# B&R Automation Studio project mappFramework (part 2)

### SimpleCfg.mpreportcore - PC/mappServices/Report/SimpleCfg.mpreportcore
```
Element gMpLinkSimpleReport (Type=mpreportcore)
  MpReport:
    Settings:
      ResourceDeviceName = mappReportFiles
      LanguageDependent:
        [0]:
          Language = en
        [1]:
          Language = de
        [2]:
          Language = zh
    PageLayouts:
      [0]:
        Name = Default
        Orientation = 2
        Margins = 2
    Styles:
      Text:
        [0]:
          Name = Default
        [1]:
          Name = Title
          Size = 20
        [2]:
          Name = Description
          Color = FF9900
        [3]:
          Name = TableText
          NumberOfDecimalPlaces = 2
        [4]:
          Name = ChartText
          NumberOfDecimalPlaces = 2
      Table:
        [0]:
          Name = Default
        [1]:
          Name = ThickBorder_Blue_HighPadding
          BorderWidth = 3
          Color = 0000FF
          Padding = 3
      Line:
        [0]:
          Name = Default
        [1]:
          Name = ThickOrangeLine
          Width = 5
          Color = FF9900
      Chart:
        PieChart:
          [0]:
            Name = Default
          [1]:
            Name = ColorPieChart
            BackColor = 008080
            BorderWidth = 3
            BorderColor = 33CC00
            Padding = 3
        LineChart:
          [0]:
            Name = Default
          [1]:
            Name = ColorLineChart
            BackColor = 008080
            BorderWidth = 3
            BorderColor = 33CC00
            Padding = 3
            GraphBackColor = C0C0C0
            GraphBorderWidth = 3
            GraphBorderColor = 808000
            GridLineWidth = 3
            GridLineColor = 7F7F7F
        BarChart:
          [0]:
            Name = Default
          [1]:
            Name = ColorBarChart
            BackColor = 008080
            BorderWidth = 3
            BorderColor = 33CC00
            Padding = 3
            ItemGapWidth = 3
            GraphBackColor = C0C0C0
            GraphBorderWidth = 3
            GraphBorderColor = 808000
            GridLineWidth = 3
            GridLineColor = 7F7F7F
    Tables:
      [0]:
        Name = DailySummary
        TableStyle = Default
        TextStyle = TableText
        [0]:
          [0] = TextId
            Source = {$mappFramework/Report/Texts/RunTime}
            Width = 20
            HorizontalAlign = 1
          [1] = TextId
            Source = {$mappFramework/Report/Texts/UpTime}
            Width = 20
            HorizontalAlign = 1
          [2] = TextId
            Source = {$mappFramework/Report/Texts/DownTime}
            Width = 20
            HorizontalAlign = 1
          [3] = TextId
            Source = {$mappFramework/Report/Texts/PartsMade}
            Width = 20
            HorizontalAlign = 1
          [4] = TextId
            Source = {$mappFramework/Report/Texts/PPM}
            Width = 10
            HorizontalAlign = 1
          [5] = TextId
            Source = {$mappFramework/Report/Texts/NumRejects}
            Width = 10
            HorizontalAlign = 1
        [1]:
          [0] = ValueId
            Value:
              ProcessVariable = ::ReportMgr:ReportExample.SimpleReport.OeeLine[0].RunTime
            Width = 20
          [1] = ValueId
            Value:
              ProcessVariable = ::ReportMgr:ReportExample.SimpleReport.OeeLine[0].UpTime
            Width = 20
          [2] = ValueId
            Value:
              ProcessVariable = ::ReportMgr:ReportExample.SimpleReport.OeeLine[0].DownTime
            Width = 20
          [3] = ValueId
            Value:
              ProcessVariable = ::ReportMgr:ReportExample.SimpleReport.OeeLine[0].PartsMade
            Width = 20
            HorizontalAlign = 2
          [4] = ValueId
            Value:
              ProcessVariable = ::ReportMgr:ReportExample.SimpleReport.OeeLine[0].PPM
            Width = 10
            HorizontalAlign = 2
          [5] = ValueId
            Value:
              ProcessVariable = ::ReportMgr:ReportExample.SimpleReport.OeeLine[0].NumRejects
            Width = 10
            HorizontalAlign = 2
        [2]:
          [0] = ValueId
            Value:
              ProcessVariable = ::ReportMgr:ReportExample.SimpleReport.OeeLine[1].RunTime
            Width = 20
          [1] = ValueId
            Value:
              ProcessVariable = ::ReportMgr:ReportExample.SimpleReport.OeeLine[1].UpTime
            Width = 20
          [2] = ValueId
            Value:
              ProcessVariable = ::ReportMgr:ReportExample.SimpleReport.OeeLine[1].DownTime
            Width = 20
          [3] = ValueId
            Value:
              ProcessVariable = ::ReportMgr:ReportExample.SimpleReport.OeeLine[1].PartsMade
            Width = 20
            HorizontalAlign = 2
          [4] = ValueId
            Value:
              ProcessVariable = ::ReportMgr:ReportExample.SimpleReport.OeeLine[1].PPM
            Width = 10
            HorizontalAlign = 2
          [5] = ValueId
            Value:
              ProcessVariable = ::ReportMgr:ReportExample.SimpleReport.OeeLine[1].NumRejects
            Width = 10
            HorizontalAlign = 2
        [3]:
          [0] = ValueId
            Value:
              ProcessVariable = ::ReportMgr:ReportExample.SimpleReport.OeeLine[2].RunTime
            Width = 20
          [1] = ValueId
            Value:
              ProcessVariable = ::ReportMgr:ReportExample.SimpleReport.OeeLine[2].UpTime
            Width = 20
          [2] = ValueId
            Value:
              ProcessVariable = ::ReportMgr:ReportExample.SimpleReport.OeeLine[2].DownTime
            Width = 20
          [3] = ValueId
            Value:
              ProcessVariable = ::ReportMgr:ReportExample.SimpleReport.OeeLine[2].PartsMade
            Width = 20
            HorizontalAlign = 2
          [4] = ValueId
            Value:
              ProcessVariable = ::ReportMgr:ReportExample.SimpleReport.OeeLine[2].PPM
            Width = 10
            HorizontalAlign = 2
          [5] = ValueId
            Value:
              ProcessVariable = ::ReportMgr:ReportExample.SimpleReport.OeeLine[2].NumRejects
            Width = 10
            HorizontalAlign = 2
    Charts:
      [0] = LineChart
        Name = TempLineChart
        Heading = SingleText
          Text = {$mappFramework/Report/Texts/TempLineChartHeading}
          HorizontalAlign = 1
          TextStyle = Default
        ChartStyle = Default
        TextStyle = ChartText
        ShowLegend = 4
        Y[0]:
          Name = Temperature
          Label = {$mappFramework/Report/Texts/TempChartYAxisLabel}
          NumberOfGridLines = 9
          GraphMinValue:
            Value = 10
          GraphMaxValue:
            Value = 110
        XAxis:
          ProcessVariable = ::ReportMgr:ReportExample.SimpleReport.OeeLine[0].TemperatureSample.TimeStamp
        [0]:
          YAxis = Temperature
          Value:
            ProcessVariable = ::ReportMgr:ReportExample.SimpleReport.OeeLine[0].TemperatureSample.Value
          LegendText = {$mappFramework/Report/Texts/Line1LegendText}
        [1]:
          YAxis = Temperature
          Value:
            ProcessVariable = ::ReportMgr:ReportExample.SimpleReport.OeeLine[1].TemperatureSample.Value
          LineColor = 33CC00
          LegendText = {$mappFramework/Report/Texts/Line2LegendText}
        [2]:
          YAxis = Temperature
          Value:
            ProcessVariable = ::ReportMgr:ReportExample.SimpleReport.OeeLine[2].TemperatureSample.Value
          LineColor = 0000FF
          LegendText = {$mappFramework/Report/Texts/Line3LegendText}
      [1] = BarChart
        Name = PartsBarChart
        ChartStyle = Default
        TextStyle = ChartText
        ShowLegend = 4
        YAxis:
          Label = {$mappFramework/Report/Texts/PartsMade}
          NumberOfGridLines = 9
          ItemMaxValue:
            Value = 100000
        [0]:
          Value:
            ProcessVariable = ::ReportMgr:ReportExample.SimpleReport.OeeLine[0].PartsMade
          ItemColor = 0000FF
          LegendText = {$mappFramework/Report/Texts/Line1LegendText}
        [1]:
          Value:
            ProcessVariable = ::ReportMgr:ReportExample.SimpleReport.OeeLine[1].PartsMade
          ItemColor = 008080
          LegendText = {$mappFramework/Report/Texts/Line2LegendText}
        [2]:
          Value:
            ProcessVariable = ::ReportMgr:ReportExample.SimpleReport.OeeLine[2].PartsMade
          ItemColor = 33CC00
          LegendText = {$mappFramework/Report/Texts/Line3LegendText}
      [2] = BarChart
        Name = RejectsBarChart
        ChartStyle = Default
        TextStyle = ChartText
        ShowLegend = 4
        YAxis:
          Label = {$mappFramework/Report/Texts/NumRejects}
          NumberOfGridLines = 9
          ItemMaxValue:
            Value = 1500
        [0]:
          Value:
            ProcessVariable = ::ReportMgr:ReportExample.SimpleReport.OeeLine[0].NumRejects
          ItemColor = 0000FF
          LegendText = {$mappFramework/Report/Texts/Line1LegendText}
        [1]:
          Value:
            ProcessVariable = ::ReportMgr:ReportExample.SimpleReport.OeeLine[1].NumRejects
          ItemColor = 008080
          LegendText = {$mappFramework/Report/Texts/Line2LegendText}
        [2]:
          Value:
            ProcessVariable = ::ReportMgr:ReportExample.SimpleReport.OeeLine[2].NumRejects
          ItemColor = 33CC00
          LegendText = {$mappFramework/Report/Texts/Line3LegendText}
      [3]:
        Name = LineOnePie
        ChartStyle = Default
        TextStyle = ChartText
        ShowLegend = 4
        [0]:
          Value:
            ProcessVariable = ::ReportMgr:ReportExample.SimpleReport.OeeLine[0].PartsMade
          ItemBackColor = FF9900
          LegendText = {$mappFramework/Report/Texts/PartsMade}
        [1]:
          Value:
            ProcessVariable = ::ReportMgr:ReportExample.SimpleReport.OeeLine[0].NumRejects
          ItemBackColor = 7F7F7F
          LegendText = {$mappFramework/Report/Texts/NumRejects}
      [4]:
        Name = LineTwoPie
        ChartStyle = Default
        TextStyle = ChartText
        ShowLegend = 4
        [0]:
          Value:
            ProcessVariable = ::ReportMgr:ReportExample.SimpleReport.OeeLine[1].PartsMade
          ItemBackColor = FF9900
          LegendText = {$mappFramework/Report/Texts/PartsMade}
        [1]:
          Value:
            ProcessVariable = ::ReportMgr:ReportExample.SimpleReport.OeeLine[1].NumRejects
          ItemBackColor = 7F7F7F
          LegendText = {$mappFramework/Report/Texts/NumRejects}
      [5]:
        Name = LineThreePie
        ChartStyle = Default
        TextStyle = ChartText
        ShowLegend = 4
        [0]:
          Value:
            ProcessVariable = ::ReportMgr:ReportExample.SimpleReport.OeeLine[2].PartsMade
          ItemBackColor = FF9900
          LegendText = {$mappFramework/Report/Texts/PartsMade}
        [1]:
          Value:
            ProcessVariable = ::ReportMgr:ReportExample.SimpleReport.OeeLine[2].NumRejects
          ItemBackColor = 7F7F7F
          LegendText = {$mappFramework/Report/Texts/NumRejects}
    Components:
      [0]:
        AlarmHistoryLink = gMpLinkAlarmXHistory
        EmptyListText = {$mappFramework/Report/Texts/EmptyAlarmListText}
        TableStyle = Default
        TextStyle = TableText
        SELECT:
          [0]:
            Column = TimeStamp
            Width = 20
            Heading = SingleText
              Text = {$mappFramework/Report/Texts/TimeStamp}
          [1]:
            Column = Code
            Width = 5
            Heading = SingleText
              Text = {$mappFramework/Report/Texts/Code}
          [2]:
            Width = 15
            Heading = SingleText
              Text = {$mappFramework/Report/Texts/Name}
          [3]:
            Column = Message
            Width = 40
            Heading = SingleText
              Text = {$mappFramework/Report/Texts/Message}
          [4]:
            Column = StateChange
              DisplayAs:
                ActiveText = {$mappFramework/Report/Texts/Activated}
                InactiveText = {$mappFramework/Report/Texts/Deactivated}
                AcknowledgeText = {$mappFramework/Report/Texts/Acknowledged}
                UnacknowledgeText = {$mappFramework/Report/Texts/Unacknowledged}
                UpdateText = {$mappFramework/Report/Texts/Updated}
            Width = 20
            Heading = SingleText
              Text = {$mappFramework/Report/Texts/StateChange}
    Contents:
      [0]:
        Name = Header
        [0] = Image
          Image = Images\LogoWithTag.jpg
          HorizontalAlign = 2
        [1]:
          Text = {$mappFramework/Report/Texts/SimpleHeaderText}
          HorizontalAlign = 1
          NewLine = FALSE
          TextStyle = Title
        [2] = EmptyLine
          Size = 20
      [1]:
        Name = Footer
        [0] = PageNumber
          PageNumSnippet = {$mappFramework/Report/Texts/FooterText}
          HorizontalAlign = 2
          NewLine = FALSE
          TextStyle = Description
      [2]:
        Name = Intro
        [0]:
          Text = {$mappFramework/Report/Texts/IntroText}
          TextStyle = Default
        [1] = EmptyLine
          Size = 20
      [3]:
        Name = DailySummary
        [0] = Line
          LineStyle = Default
        [1] = EmptyLine
          Size = 20
        [2]:
          Text = {$mappFramework/Report/Texts/DailySummaryText}
          HorizontalAlign = 1
          TextStyle = Description
        [3] = EmptyLine
          Size = 20
        [4] = Table
          Table = DailySummary
          HorizontalAlign = 1
        [5] = EmptyLine
          Size = 20
      [4]:
        Name = ProductsChart
        [0] = Line
          LineStyle = Default
        [1] = EmptyLine
          Size = 20
        [2]:
          Text = {$mappFramework/Report/Texts/ProductsChartText}
          HorizontalAlign = 1
          TextStyle = Description
        [3] = EmptyLine
          Size = 20
        [4] = Chart
          Chart = PartsBarChart
          Width = 60
          Height = UserDefined
            Scaling = 35
          HorizontalAlign = 1
        [5] = EmptyLine
          Size = 20
      [5]:
        Name = RejectsChart
        [0]:
          Text = {$mappFramework/Report/Texts/RejectsChartText}
          HorizontalAlign = 1
          TextStyle = Description
        [1] = EmptyLine
          Size = 20
        [2] = Chart
          Chart = RejectsBarChart
          Width = 60
          Height = UserDefined
            Scaling = 35
          HorizontalAlign = 1
        [3] = EmptyLine
          Size = 20
      [6]:
        Name = LineOnePie
        [0]:
          Text = {$mappFramework/Report/Texts/Line1PieText}
          HorizontalAlign = 1
          TextStyle = Description
        [1] = Chart
          Chart = LineOnePie
          Width = 60
          Height = UserDefined
            Scaling = 28
          HorizontalAlign = 1
        [2] = EmptyLine
          Size = 20
      [7]:
        Name = LineTwoPie
        [0]:
          Text = {$mappFramework/Report/Texts/Line2PieText}
          HorizontalAlign = 1
          TextStyle = Description
        [1] = Chart
          Chart = LineTwoPie
          Width = 60
          Height = UserDefined
            Scaling = 28
          HorizontalAlign = 1
        [2] = EmptyLine
          Size = 20
      [8]:
        Name = LineThreePie
        [0]:
          Text = {$mappFramework/Report/Texts/Line3PieText}
          HorizontalAlign = 1
          TextStyle = Description
        [1] = Chart
          Chart = LineThreePie
          Width = 60
          Height = UserDefined
            Scaling = 28
          HorizontalAlign = 1
      [9]:
        Name = TemperatureChart
        [0] = Line
          LineStyle = Default
        [1] = EmptyLine
          Size = 20
        [2]:
          Text = {$mappFramework/Report/Texts/TempChartText}
          HorizontalAlign = 1
          TextStyle = Description
        [3] = EmptyLine
          Size = 20
        [4] = Chart
          Chart = TempLineChart
          Height = UserDefined
            Scaling = 80
          HorizontalAlign = 1
        [5] = EmptyLine
          Size = 20
      [10]:
        Name = Alarms
        [0] = Line
          LineStyle = Default
        [1] = Component
          Component = AlarmHistory
        [2] = EmptyLine
          Size = 20
      [11]:
        Name = Audits
        [0] = Line
          LineStyle = Default
        [1] = Component
          Component = AuditTrail
        [2] = EmptyLine
          Size = 20
    Reports:
      [0]:
        Name = SimpleReport
        PageLayout = Default
        Header = Header
        Footer = Footer
        [0]:
          Heading:
            Text = 
            HorizontalAlign = 1
            TextStyle = Default
          [0]:
            Content = Intro
        [1]:
          Heading:
            Text = {$mappFramework/Report/Texts/DailySummaryHeading}
            TextStyle = Default
          [0]:
            Content = DailySummary
        [2]:
          StartOnNewPage = TRUE
          Heading:
            Text = {$mappFramework/Report/Texts/PartsAndRejectsHeading}
            TextStyle = Default
          [0]:
            Content = ProductsChart
        [3]:
          [0]:
            Content = RejectsChart
        [4]:
          StartOnNewPage = TRUE
          Heading:
            Text = {$mappFramework/Report/Texts/PartsAndRejectsHeading}
            TextStyle = Default
          [0]:
            Content = LineOnePie
        [5]:
          Heading:
            Text = 
            TextStyle = Default
          [0]:
            Content = LineTwoPie
        [6]:
          Heading:
            Text = 
            TextStyle = Default
          [0]:
            Content = LineThreePie
        [7]:
          StartOnNewPage = TRUE
          Heading:
            Text = {$mappFramework/Report/Texts/TempSamplesHeading}
            TextStyle = Default
          [0]:
            Content = TemperatureChart
        [8]:
          StartOnNewPage = TRUE
          Heading:
            Text = {$mappFramework/Report/Texts/AlarmHeading}
            TextStyle = Default
          [0]:
            Content = Alarms
  Alarms = MpAlarmX
    mapp.AlarmX.Core.Configuration:
      [0]:
        Message = {$mappFramework/Report/Alarms/GenerateFailed}
```

### UserXCfg.mpuserx - PC/mappServices/UserX/UserXCfg.mpuserx
```
Element UserMgmtX (Type=mpuserx)
  Mgr:
    PasswordChangeInterval = 7776000
    PasswordExpirationNotification = 864000
    UserExpirationTime = 31536000
    PasswordAlpha = TRUE
    PasswordLength = 6
    UserNameLength = 3
    LoginAttempts = 5
  ServerSettings:
    Server:
      AdditionalUserData:
        [0] = mail
        [1] = telephoneNumber
  Users:
    DefUser#1:
      id = Admin
      name = Admin
      lang = en
      unit = imperial
    DefUser#2:
      id = Anonymous
      name = Anonymous
      lang = en
      unit = metric
    DefUser#3:
      id = Operator
      name = Operator
      lang = en
      unit = imperial-us
    DefUser#4:
      id = Service_Tech
      name = Service_Tech
      lang = zh
      unit = metric
  Groups:
    DefGroup#1:
      id = Administrators
      level = 100
      admin = TRUE
      rights:
        [0] = FullAccess
        [1] = ViewOnly
        [2] = StartOnly
    DefGroup#2:
      id = Everyone
      level = 3
      rights:
        [0] = ViewOnly
    DefGroup#3:
      id = Operators
      level = 30
      rights:
        [0] = StartOnly
    DefGroup#4:
      id = Service
      level = 50
      rights:
        [0] = StartOnly
        [1] = ViewOnly
```

### UserXlogin.mpuserxlogin - PC/mappServices/UserX/UserXlogin.mpuserxlogin
```
Element gMpLinkUserXLogin (Type=mpuserxlogin)
  Alarms = MpAlarmX
    mapp.AlarmX.Core.Configuration:
      [0]:
        Message = {$UserX/Alarms/UserLocked}
```

## Configuration SimulationVC4

CPU PC_any, AutomationRuntime E4.91, Build 6.3.0, Safety 0.0, Vc V4.72.3

### Task classes (Cpu.sw)
```
Cyclic#1 (cycle 10000 us):
  AlarmMgr <- Infrastructure.VC4.AlarmX.AlarmMgr.prg
  AppAxis_1 <- MachineControl.AppAxis_1.AppAxis_1.prg
  AxisMgr <- MachineControl.AxisTemplate.AxisMgr.prg [disabled]
Cyclic#8 (cycle 10000 us):
  BackupMgr <- Infrastructure.VC4.Backup.BackupMgr.prg
  FileMgr <- Infrastructure.VC4.File.FileMgr.prg
  UsbMgr <- Infrastructure.VC4.Usb.UsbMgr.prg  // USB manager
  RecipeMgr <- Infrastructure.VC4.Recipe.RecipeMgr.prg
  UserXMgr <- Infrastructure.VC4.UserX.UserXMgr.prg
  AuditMgr <- Infrastructure.VC4.Audit.AuditMgr.prg
  ReportMgr <- Infrastructure.VC4.Report.ReportMgr.prg
NcDataObjects: McDriveLog
VcDataObjects: mappFr <- VC4.mappFrameworkVisu.dob
Binaries: arsvcreg, mCoWebSc, McProfGen, mcacpdrv, TCLang, arflatprv, FWRules, arcoal, udbdef, mvLoader, TCData, MachineGrp, UserXCfg, UserXlogin, arconfig, FileCfg, RecipeXML, TC, RecipeFile, User, AlarmXCfg, asfw, iomap, Role, Axis1Alm, VAppAxis1, ashwd, RecipeCSV, Settings, AppAxis1, BackupCfg, ashwac, AlarmXHist, sysconf, Axis1Grp, BackupFile, AuditCfg, UnitCfg, CustomCfg
Libraries: runtime, astime, FileIO, AsBrStr, MpBase, MpAlarmX, MpServer, sys_lib, standard, AsZip, CoTrace, MpAxis, MpRecipe, MpCom, McAxis, McBase, McAcpAx, McPureVAx, McAcpPar, AsIODiag, MpFile, MpBackup, AsUSB, MpUserX, AsARCfg, IecCheck, MpAudit, MpReport, asieccon, brsystem, aseth, ashw, powerlnk, dataobj, arssl, arproject, arcert, aruser, asepl
```

### Hardware
```
PC : PC_any v1.1.1.0 (OrderNumber=PC)
  Connector IF3:
    Vnc1
    VncVcObjectName1 = mappFr
    VncKeyMappingFile1 = VC\PS2-Keyboard.dis
  ConfigurationID = mappFramework516_Simulation
  UserPartitionSize = 256
  Cyclic1Duration = 10000
  Cyclic1Stack = 32000
  Cyclic5Duration = 10000
  Cyclic8Duration = 10000
  Cyclic8Stack = 32000
  FileDevice1
  FileDeviceName1 = USER
  FileDevicePath1 = USER_PATH
  FileDevice2
  FileDeviceName2 = mappAlarmXFiles
  FileDevicePath2 = USER_PATH:\AlarmX
  FileDevice3
  FileDeviceName3 = mappBackupFiles
  FileDevicePath3 = USER_PATH:\Backup
  FileDevice4
  FileDeviceName4 = mappRecipeFiles
  FileDevicePath4 = USER_PATH:\Recipe
  FileDevice5
  FileDeviceName5 = mappUserXFiles
  FileDevicePath5 = USER_PATH:\UserX
  FileDevice6
  FileDeviceName6 = mappAuditFiles
  FileDevicePath6 = USER_PATH:\Audit
  FileDevice7
  FileDeviceName7 = mappDataFiles
  FileDevicePath7 = USER_PATH:\Data
  FileDevice8
  FileDeviceName8 = mappReportFiles
  FileDevicePath8 = USER_PATH:\Report
  FtpUser1
  FtpUsername1 = Admin
  FtpUserPassword1 = jhTZ9rja+dMo4uQziZxIvYZJ7RF3iWJ9y9zyiFMZfoo=  // 123ABc
  FtpUserSalt1 = 8r0jnJ0m
  FTPAccessRight1 = 0
  FTPdevice1 = ALL
  ActivateOpcUa = 1
  OpcUaActivateAuditEvents = 1
  OpcUa_Security_AdminRole = Administrators
  OpcUaInformationModels_PV_Version = 1
```

### PackMLCfg.mppackmlcore - PC/mappServices/PackML/PackMLCfg.mppackmlcore
```
Element gMpLinkPackMLCore (Type=mppackmlcore)
  Modes:
    Mode[1]:
      ModeID = 1
      Name = Production
  Unit:
    StartupActiveMode = 1
    ResetCommands = 1
  UnitModes:
    Mode[1]:
      ModeID = 1
      Name = Automatic Mode
    Mode[2]:
      ModeID = 2
      State[5] = 0
      State[17] = 0
    Mode[3]:
      ModeID = 3
      State[1] = 0
      State[5] = 0
      State[11] = 0
      State[17] = 0
  Alarms = MpAlarmX
    mapp.AlarmX.Core.Configuration:
      [0]:
        Message = {$mappFramework/PackML/Alarms/StateTransitionNotAllowed}
      [1]:
        Message = {$mappFramework/PackML/Alarms/ModeTransitionNotAllowed}
      [2]:
        Message = {$mappFramework/PackML/Alarms/ConfigurationInvalid}
```

### PackMLMain.mppackmlmodule - PC/mappServices/PackML/PackMLMain.mppackmlmodule
```
Element gPackMLModule_Main (Type=mppackmlmodule)
  Module:
    Name = Main
    Parent = 1
      Unit = gMpLinkPackMLCore
      Activation = 0
```

## Configuration SourceReference

CPU PC_any, AutomationRuntime E4.91, Build 6.3.0, Safety 0.0, Vc 

### Task classes (Cpu.sw)
```
Cyclic#1 (cycle 10000 us):
  AlarmMgr <- Infrastructure.AlarmX.AlarmMgr.prg
  AppAxis_1 <- MachineControl.AppAxis_1.AppAxis_1.prg
  AxisMgr <- MachineControl.AxisTemplate.AxisMgr.prg [disabled]
Cyclic#8 (cycle 10000 us):
  BackupMgr <- Infrastructure.Backup.BackupMgr.prg
  FileMgr <- Infrastructure.File.FileMgr.prg
  UsbMgr <- Infrastructure.Usb.UsbMgr.prg  // USB manager
  RecipeMgr <- Infrastructure.Recipe.RecipeMgr.prg
  UserXMgr <- Infrastructure.UserX.UserXMgr.prg
  AuditMgr <- Infrastructure.Audit.AuditMgr.prg
  ReportMgr <- Infrastructure.Report.ReportMgr.prg
NcDataObjects: McDriveLog
Binaries: arsvcreg, mCoWebSc, McProfGen, mcacpdrv, TCLang, arflatprv, FWRules, arcoal, udbdef, mvLoader, TCData, MachineGrp, UserXCfg, UserXlogin, arconfig, FileCfg, RecipeXML, TC, RecipeFile, User, AlarmXCfg, asfw, iomap, Role, Axis1Alm, VAppAxis1, ashwd, RecipeCSV, Settings, AppAxis1, BackupCfg, ashwac, AlarmXHist, sysconf, Axis1Grp, BackupFile, AuditCfg, UnitCfg, CustomCfg
Libraries: runtime, astime, FileIO, AsBrStr, MpBase, MpAlarmX, MpServer, sys_lib, standard, AsZip, CoTrace, MpAxis, MpRecipe, MpCom, McAxis, McBase, McAcpAx, McPureVAx, McAcpPar, AsIODiag, MpFile, MpBackup, AsUSB, MpUserX, AsARCfg, IecCheck, MpAudit, MpReport, asieccon, brsystem, aseth, ashw, powerlnk, dataobj, arssl, arproject, arcert, aruser, asepl
```

### Hardware
```
PC : PC_any v1.1.1.0 (OrderNumber=PC)
  ConfigurationID = mappFramework516_Simulation
  UserPartitionSize = 256
  Cyclic1Duration = 10000
  Cyclic1Stack = 32000
  Cyclic5Duration = 10000
  Cyclic8Duration = 10000
  Cyclic8Stack = 32000
  FileDevice1
  FileDeviceName1 = UserPartition
  FileDevicePath1 = USER_PATH
  FileDevice2
  FileDeviceName2 = mappAlarmXFiles
  FileDevicePath2 = USER_PATH:\AlarmX
  FileDevice3
  FileDeviceName3 = mappBackupFiles
  FileDevicePath3 = USER_PATH:\Backup
  FileDevice4
  FileDeviceName4 = mappRecipeFiles
  FileDevicePath4 = USER_PATH:\Recipe
  FileDevice5
  FileDeviceName5 = mappUserXFiles
  FileDevicePath5 = USER_PATH:\UserX
  FileDevice6
  FileDeviceName6 = mappAuditFiles
  FileDevicePath6 = USER_PATH:\Audit
  FileDevice7
  FileDeviceName7 = mappDataFiles
  FileDevicePath7 = USER_PATH:\Data
  FileDevice8
  FileDeviceName8 = mappReportFiles
  FileDevicePath8 = USER_PATH:\Report
  FtpUser1
  FtpUsername1 = Admin
  FtpUserPassword1 = jhTZ9rja+dMo4uQziZxIvYZJ7RF3iWJ9y9zyiFMZfoo=  // 123ABc
  FtpUserSalt1 = 8r0jnJ0m
  FTPAccessRight1 = 0
  FTPdevice1 = ALL
  ActivateOpcUa = 1
  OpcUaInformationModels_PV_Version = 1
```

## Configuration UnitTest

CPU , AutomationRuntime E4.91, Build 6.3.0, Safety 0.0

### Task classes (Cpu.sw)
```
Cyclic#1 (cycle 10000 us):
  AppAxis_1 <- MachineControl.AppAxis_1.AppAxis_1.prg
Cyclic#8 (cycle 10000 us):
  AlarmMgr <- Infrastructure.VC4.AlarmX.AlarmMgr.prg
  AlarmXUnit <- UnitTest.AlarmX.AlarmXUnitTest.prg
  AuditMgr <- Infrastructure.VC4.Audit.AuditMgr.prg
  AuditTest <- UnitTest.Audit.AuditTest.prg
  BackupMgr <- Infrastructure.VC4.Backup.BackupMgr.prg
  BackupUnit <- UnitTest.Backup.BackupUnitTest.prg
  UsbMgr <- Infrastructure.VC4.Usb.UsbMgr.prg
  RecipeMgr <- Infrastructure.VC4.Recipe.RecipeMgr.prg
  RecipeMgrU <- UnitTest.Recipe.RecipeMgrUnitTest.prg
  UserXMgr <- Infrastructure.VC4.UserX.UserXMgr.prg
  UserXUnitT <- UnitTest.UserX.UserXUnitTest.prg
  FileMgr <- Infrastructure.VC4.File.FileMgr.prg
  FileTest <- UnitTest.File.FileUnitTest.prg
  AppAxisUni <- UnitTest.AppAxis_1.AppAxisUnitTest.prg
  ReportUnit <- UnitTest.Report.ReportUnitTest.prg
  ReportMgr <- Infrastructure.VC4.Report.ReportMgr.prg
NcDataObjects: mcdrivelog
Binaries: arsvcreg, TCData, TCLang, mvLoader, udbdef, mCoWebSc, arcoal, arflatprv, mcprofgen, mcacpdrv, asfw, ashwd, ashwac, iomap, arconfig, sysconf, FileCfg, RecipeFile, Axis1Grp, Axis1Alm, AlarmXCfg, UserXCfg, BackupCfg, AlarmXHist, UserXlogin, BackupFile, RecipeCSV, RecipeXML, TC, UnitCfg, CustomCfg, AuditCfg, MachineGrp
Libraries: Runtime, sys_lib, AsIecCon, astime, AsARCfg, AsBrStr, UnitTest, LibAssert1, UtWs, UtMgr, SPLMyCalc, snprintf, IecCheck, McBase, MpAxis, McPureVAx, McAcpPar, McAcpAx, McAxis, MpBase, ArTextSys, standard, operator, AsBrWStr, asusb, mpfile, fileio, arssl, arproject, mprecipe, asepl, mpuserx, arcert, mpbackup, ashw, asiodiag, aruser, dataobj, mpalarmx, aseth, powerlnk, brsystem, mpaudit
```

### Hardware
```
PC_any : PC_any v1.1.1.0 (OrderNumber=PC)
  ConfigurationID = mappFramework_UnitTest
  UserPartitionSize = 256
  AutomaticTransferOfUserfiles = on
  Cyclic1Duration = 10000
  Cyclic4Duration = 10000
  Cyclic8Duration = 10000
  FileDevice1
  FileDeviceName1 = USER
  FileDevicePath1 = USER_PATH
  FileDevice2
  FileDeviceName2 = mappAlarmXFiles
  FileDevicePath2 = USER_PATH\AlarmX
  FileDevice3
  FileDeviceName3 = mappAuditFiles
  FileDevicePath3 = USER_PATH\Audit
  FileDevice4
  FileDeviceName4 = mappBackupFiles
  FileDevicePath4 = USER_PATH\Backup
  FileDevice5
  FileDeviceName5 = mappDataFiles
  FileDevicePath5 = USER_PATH\Data
  FileDevice6
  FileDeviceName6 = mappRecipeFiles
  FileDevicePath6 = USER_PATH\Recipe
  FileDevice7
  FileDeviceName7 = mappUserXFiles
  FileDevicePath7 = USER_PATH\UserX
  FileDevice8
  FileDeviceName8 = mappReportFiles
  FileDevicePath8 = USER_PATH\Report
```

### File.vvm - PC_any/File.vvm
```iecst
VAR_CONFIG
	::FileTest:HmiFile_UT.Parameters AT %Q.::FileMgr:HmiFile.Parameters; (*Insert your comment here...*)
	::FileMgr:HmiFile.Status AT %Q.::FileTest:HmiFile_UT.Status; (*Insert your comment here...*)
END_VAR
```

### AlarmMgr.vvm - PC_any/UnitTest/AlarmMgr.vvm
```iecst
(*Inputs to the unit test*)
VAR_CONFIG
	::AlarmMgr:MpAlarmXCore_0.StatusID AT %Q.::AlarmXUnit:MpBlockStatus[0]; (*Insert your comment here...*)
	::AlarmMgr:MpAlarmXHistory_0.StatusID AT %Q.::AlarmXUnit:MpBlockStatus[1]; (*Insert your comment here...*)
	::AlarmMgr:MpAlarmXHistoryUI_0.StatusID AT %Q.::AlarmXUnit:MpBlockStatus[2]; (*Insert your comment here...*)
	::AlarmMgr:MpAlarmXControlExample_0.StatusID AT %Q.::AlarmXUnit:MpBlockStatus[3]; (*Insert your comment here...*)
	::AlarmMgr:MpAlarmXListUI_0.StatusID AT %Q.::AlarmXUnit:MpBlockStatus[4]; (*Insert your comment here...*)
	::AlarmMgr:QueryActiveAlarms_0.StatusID AT %Q.::AlarmXUnit:MpBlockStatus[5]; (*Insert your comment here...*)
	::AlarmMgr:MpAlarmXCore_0 AT %Q.::AlarmXUnit:MpAlarmXCore_0; (*Insert your comment here...*)
	::AlarmMgr:MpAlarmXListUIConnect AT %Q.::AlarmXUnit:MpAlarmXListUIConnect; (*Insert your comment here...*)
END_VAR
(*Outputs from the unit test*)
VAR_CONFIG
	::AlarmXUnit:AlarmExamples AT %Q.::AlarmMgr:AlarmExamples; (*Insert your comment here...*)
END_VAR
```

### AppAxis.vvm - PC_any/UnitTest/AppAxis.vvm
```iecst
(*Inputs to the unit test*)
VAR_CONFIG
	::AppAxis_1:MpAxisBasic_0.StatusID AT %Q.::AppAxisUni:MpBlockStatus[0]; (*Insert your comment here...*)
	::AppAxis_1:MpAlarmXCore_0.StatusID AT %Q.::AppAxisUni:MpBlockStatus[1]; (*Insert your comment here...*)
	::AppAxis_1:MpRecipeRegPar_Cfg.StatusID AT %Q.::AppAxisUni:MpBlockStatus[2]; (*Insert your comment here...*)
	::AppAxis_1:MpRecipeRegPar_Par.StatusID AT %Q.::AppAxisUni:MpBlockStatus[3]; (*Insert your comment here...*)
	::AppAxis_1:AxisControl.Status AT %Q.::AppAxisUni:AxisControl.Status; (*Insert your comment here...*)
	::AppAxis_1:MpAlarmXCore_0 AT %Q.::AppAxisUni:MpAlarmXCore_0; (*Insert your comment here...*)
	::AppAxis_1:State AT %Q.::AppAxisUni:State; (*Insert your comment here...*)
END_VAR
(*Outputs from the unit test*)
VAR_CONFIG
	::AppAxisUni:AxisControl.Command AT %Q.::AppAxis_1:AxisControl.Command; (*Insert your comment here...*)
	::AppAxisUni:AxisControl.Parameters AT %Q.::AppAxis_1:AxisControl.Parameters; (*Insert your comment here...*)
END_VAR
```

### AuditMgr.vvm - PC_any/UnitTest/AuditMgr.vvm
```iecst
(*Inputs to the unit test*)
VAR_CONFIG
	::AuditMgr:MpAuditTrail_0.CommandDone AT %Q.::AuditTest:MpAuditTrailCmdDone; (*Insert your comment here...*)
	::AuditMgr:HmiAudit.Status.ArchiveAvailable AT %Q.::AuditTest:HmiAudit.Status.ArchiveAvailable; (*Insert your comment here...*)
	::AuditMgr:HmiAudit.Status.NumberOfArchives AT %Q.::AuditTest:HmiAudit.Status.NumberOfArchives; (*Insert your comment here...*)
	::AuditMgr:MpAuditTrail_0.Error AT %Q.::AuditTest:MpAuditTrailError; (*Insert your comment here...*)
END_VAR
(*Outputs from the unit test*)
VAR_CONFIG
	::AuditTest:HmiAudit.Commands.ExportArchives AT %Q.::AuditMgr:HmiAudit.Commands.ExportArchives; (*Insert your comment here...*)
	::AuditTest:SampleTemperature AT %Q.::AuditMgr:VariableMonitorExample; (*Insert your comment here...*)
	::AuditTest:HmiAudit.Parameters.ArchiveSettings.Enable AT %Q.::AuditMgr:HmiAudit.Parameters.ArchiveSettings.Enable; (*Insert your comment here...*)
	::AuditTest:HmiAudit.Parameters.ArchiveSettings.MaxSize AT %Q.::AuditMgr:HmiAudit.Parameters.ArchiveSettings.MaxSize; (*Insert your comment here...*)
	::AuditTest:HmiAudit.Parameters.ArchiveSettings.Mode AT %Q.::AuditMgr:HmiAudit.Parameters.ArchiveSettings.Mode; (*Insert your comment here...*)
	::AuditTest:HmiAudit.Parameters.ArchiveSettings.Hour AT %Q.::AuditMgr:HmiAudit.Parameters.ArchiveSettings.Hour; (*Insert your comment here...*)
	::AuditTest:HmiAudit.Parameters.ArchiveSettings.Minute AT %Q.::AuditMgr:HmiAudit.Parameters.ArchiveSettings.Minute; (*Insert your comment here...*)
	::AuditTest:HmiAudit.Parameters.ArchiveSettings.FileType AT %Q.::AuditMgr:HmiAudit.Parameters.ArchiveSettings.FileType; (*Insert your comment here...*)
END_VAR
```

### BackupMgr.vvm - PC_any/UnitTest/BackupMgr.vvm
```iecst
VAR_CONFIG
	::BackupMgr:MpBackupCoreSys.StatusID AT %Q.::BackupUnit:MpBlockStatus[0]; (*Insert your comment here...*)
	::BackupMgr:MpBackupCoreConfigSys.StatusID AT %Q.::BackupUnit:MpBlockStatus[1]; (*Insert your comment here...*)
	::BackupMgr:MpFileManagerUIBackup.StatusID AT %Q.::BackupUnit:MpBlockStatus[2]; (*Insert your comment here...*)
END_VAR
```

### File.vvm - PC_any/UnitTest/File.vvm
```iecst
VAR_CONFIG
	Cyclic#8.::FileTest:HmiFile_UT.Parameters AT %Q.Cyclic#8.::FileMgr:HmiFile.Parameters; (*Insert your comment here...*)
	Cyclic#8.::FileMgr:HmiFile.Status AT %Q.Cyclic#8.::FileTest:HmiFile_UT.Status; (*Insert your comment here...*)
END_VAR
```

### FileMgr.vvm - PC_any/UnitTest/FileMgr.vvm
```iecst
(*Inputs to the unit test*)
VAR_CONFIG
	::FileMgr:MpFileManagerUISys.StatusID AT %Q.::FileTest:MpBlockStatus[0]; (*Insert your comment here...*)
	::FileMgr:MpFileManagerUI_FIFO.StatusID AT %Q.::FileTest:MpBlockStatus[1]; (*Insert your comment here...*)
	Cyclic#8.::FileMgr:HmiFile.Status AT %Q.Cyclic#8.::FileTest:HmiFile_UT.Status; (*Insert your comment here...*)
END_VAR
(*Outputs from the unit test*)
VAR_CONFIG
	Cyclic#8.::FileTest:HmiFile_UT.Parameters AT %Q.Cyclic#8.::FileMgr:HmiFile.Parameters; (*Insert your comment here...*)
	::FileTest:HmiFile.Status.SelectedIndex AT %Q.::FileMgr:HmiFile.Status.SelectedIndex; (*Insert your comment here...*)
	::FileTest:HmiFile.Commands.EnterFolder AT %Q.::FileMgr:HmiFile.Commands.EnterFolder; (*Insert your comment here...*)
	::FileTest:HmiFile.Commands.FolderUp AT %Q.::FileMgr:HmiFile.Commands.FolderUp; (*Insert your comment here...*)
END_VAR
```

### RecipeMgr.vvm - PC_any/UnitTest/RecipeMgr.vvm
```iecst
(*Inputs to the unit test*)
VAR_CONFIG
	::RecipeMgr:MpFileManagerUIRecipe.StatusID AT %Q.::RecipeMgrU:MpBlockStatus[0]; (*Insert your comment here...*)
	::RecipeMgr:MpRecipeSys.StatusID AT %Q.::RecipeMgrU:MpBlockStatus[1]; (*Insert your comment here...*)
	::RecipeMgr:MpRecipeRegPar_PreviewCfg.StatusID AT %Q.::RecipeMgrU:MpBlockStatus[2]; (*Insert your comment here...*)
	::RecipeMgr:MpRecipeRegPar_PreviewPar.StatusID AT %Q.::RecipeMgrU:MpBlockStatus[3]; (*Insert your comment here...*)
	::RecipeMgr:MpRecipeUISys.StatusID AT %Q.::RecipeMgrU:MpBlockStatus[4]; (*Insert your comment here...*)
	::RecipeMgr:MachineSettings AT %Q.::RecipeMgrU:MachineSettings; (*Insert your comment here...*)
	::RecipeMgr:Parameters AT %Q.::RecipeMgrU:Parameters; (*Insert your comment here...*)
	::RecipeMgr:HmiRecipe.Status AT %Q.::RecipeMgrU:HmiRecipe.Status; (*Insert your comment here...*)
	::RecipeMgr:MpRecipeSys AT %Q.::RecipeMgrU:MpRecipeSys; (*Insert your comment here...*)
	::RecipeMgr:MpRecipeUIConnect.Recipe.List.Names AT %Q.::RecipeMgrU:MpRecipeUIConnect.Recipe.List.Names; (*Insert your comment here...*)
	::RecipeMgr:ParametersPreview AT %Q.::RecipeMgrU:ParametersPreview; (*Insert your comment here...*)
	::RecipeMgr:MpRecipeUIConnect.Recipe.List.MaxSelection AT %Q.::RecipeMgrU:MpRecipeUIConnect.Recipe.List.MaxSelection; (*Insert your comment here...*)
	::RecipeMgr:MpRecipeUIConnect.Status AT %Q.::RecipeMgrU:MpRecipeUIConnect.Status; (*Insert your comment here...*)
	::RecipeMgr:MpRecipeUIConnect.MessageBox.LayerStatus AT %Q.::RecipeMgrU:MpRecipeUIConnect.MessageBox.LayerStatus; (*Insert your comment here...*)
END_VAR
(*Outputs from the unit test*)
VAR_CONFIG
	::RecipeMgrU:HmiRecipe.Commands AT %Q.::RecipeMgr:HmiRecipe.Commands; (*Insert your comment here...*)
	::RecipeMgrU:HmiRecipe.Parameters AT %Q.::RecipeMgr:HmiRecipe.Parameters; (*Insert your comment here...*)
	::RecipeMgrU:MpRecipeUIConnect.Recipe.Filter AT %Q.::RecipeMgr:MpRecipeUIConnect.Recipe.Filter; (*Insert your comment here...*)
	::RecipeMgrU:MpRecipeUIConnect.Recipe.Refresh AT %Q.::RecipeMgr:MpRecipeUIConnect.Recipe.Refresh; (*Insert your comment here...*)
	::RecipeMgrU:MpRecipeUIConnect.Recipe.Load AT %Q.::RecipeMgr:MpRecipeUIConnect.Recipe.Load; (*Insert your comment here...*)
	::RecipeMgrU:ParametersEdit AT %Q.::RecipeMgr:ParametersEdit; (*Insert your comment here...*)
	::RecipeMgrU:MpRecipeUIConnect.Recipe.Delete AT %Q.::RecipeMgr:MpRecipeUIConnect.Recipe.Delete; (*Insert your comment here...*)
	::RecipeMgrU:MpRecipeUIConnect.MessageBox.Confirm AT %Q.::RecipeMgr:MpRecipeUIConnect.MessageBox.Confirm; (*Insert your comment here...*)
	::RecipeMgrU:MpRecipeUIConnect.Recipe.List.SelectedIndex AT %Q.::RecipeMgr:HmiRecipe.Status.SelectedIndex; (*Insert your comment here...*)
END_VAR
```

### ReportMgr.vvm - PC_any/UnitTest/ReportMgr.vvm
```iecst
VAR_CONFIG
	::ReportMgr:MpFileManagerUI_0.StatusID AT %Q.::ReportUnit:MpBlockStatus[0]; (*Insert your comment here...*)
	Cyclic#8.::ReportUnit:HmiReport_UT.Commands AT %Q.Cyclic#8.::ReportMgr:HmiReport.Commands; (*Insert your comment here...*)
	Cyclic#8.::ReportUnit:HmiReport_UT.Parameters.UseAdvancedFormat AT %Q.Cyclic#8.::ReportMgr:HmiReport.Parameters.UseAdvancedFormat; (*Insert your comment here...*)
	Cyclic#8.::ReportMgr:HmiReport.Status AT %Q.Cyclic#8.::ReportUnit:HmiReport_UT.Status; (*Insert your comment here...*)
	Cyclic#8.::ReportMgr:MpReportCore_0.Active AT %Q.::ReportUnit:CoreInfoActive; (*Insert your comment here...*)
	Cyclic#8.::ReportMgr:MpReportCore_0.CommandDone AT %Q.::ReportUnit:CoreCmdDone; (*Insert your comment here...*)
	Cyclic#8.::ReportMgr:MpReportCore_0.Info AT %Q.::ReportUnit:CoreInfo_UT; (*Insert your comment here...*)
END_VAR
```

### UserXMgr.vvm - PC_any/UnitTest/UserXMgr.vvm
```iecst
(*Inputs to the unit test*)
VAR_CONFIG
	::UserXMgr:MpUserXLoginSys.StatusID AT %Q.::UserXUnitT:MpBlockStatus[0]; (*Insert your comment here...*)
	::UserXMgr:MpUserXLoginUISys.StatusID AT %Q.::UserXUnitT:MpBlockStatus[1]; (*Insert your comment here...*)
	::UserXMgr:MpUserXManagerUISys.StatusID AT %Q.::UserXUnitT:MpBlockStatus[2]; (*Insert your comment here...*)
END_VAR
(*Outputs from the unit test*)
```

## Configuration UnitTestVC4

CPU , AutomationRuntime E4.91, Build 6.3.0, Safety 0.0

### Task classes (Cpu.sw)
```
Cyclic#1 (cycle 10000 us):
  AppAxis_1 <- MachineControl.AppAxis_1.AppAxis_1.prg
Cyclic#8 (cycle 10000 us):
  AlarmMgr <- Infrastructure.VC4.AlarmX.AlarmMgr.prg
  AlarmXUnit <- UnitTestVC4.AlarmX.AlarmXUnitTest.prg
  AuditMgr <- Infrastructure.VC4.Audit.AuditMgr.prg
  AuditTest <- UnitTestVC4.Audit.AuditTest.prg
  BackupMgr <- Infrastructure.VC4.Backup.BackupMgr.prg
  BackupUnit <- UnitTestVC4.Backup.BackupUnitTest.prg
  UsbMgr <- Infrastructure.VC4.Usb.UsbMgr.prg
  RecipeMgr <- Infrastructure.VC4.Recipe.RecipeMgr.prg
  RecipeMgrU <- UnitTestVC4.Recipe.RecipeMgrUnitTest.prg
  UserXMgr <- Infrastructure.VC4.UserX.UserXMgr.prg
  UserXUnitT <- UnitTestVC4.UserX.UserXUnitTest.prg
  FileMgr <- Infrastructure.VC4.File.FileMgr.prg
  FileTest <- UnitTestVC4.File.FileUnitTest.prg
  AppAxisUni <- UnitTestVC4.AppAxis_1.AppAxisUnitTest.prg
  ReportUnit <- UnitTestVC4.Report.ReportUnitTest.prg
  ReportMgr <- Infrastructure.VC4.Report.ReportMgr.prg
NcDataObjects: mcdrivelog
Binaries: arsvcreg, TCData, TCLang, mvLoader, udbdef, mCoWebSc, arcoal, arflatprv, mcprofgen, mcacpdrv, FWRules, SLO_Speed, SLO_Pos, asfw, ashwd, ashwac, iomap, arconfig, sysconf, FileCfg, RecipeFile, Axis1Grp, Axis1Alm, AlarmXCfg, UserXCfg, BackupCfg, AlarmXHist, UserXlogin, BackupFile, RecipeCSV, RecipeXML, TC, UnitCfg, CustomCfg, AuditCfg, SimpleCfg, VAppAxis1, AdvCfg, Role, User, AppAxis1, ReportFile, MachineGrp
Libraries: Runtime, sys_lib, AsIecCon, astime, AsARCfg, AsBrStr, UnitTest, LibAssert1, UtWs, UtMgr, SPLMyCalc, snprintf, IecCheck, McBase, MpAxis, McPureVAx, McAcpPar, McAcpAx, McAxis, MpBase, ArTextSys, standard, operator, AsBrWStr, FileIO, AsTCP, LoggingLib, ArEventLog, asusb, mpfile, arssl, arproject, mprecipe, asepl, mpuserx, arcert, mpbackup, ashw, asiodiag, aruser, dataobj, mpalarmx, aseth, powerlnk, brsystem, mpaudit, mpreport
```

### Hardware
same as Physical/UnitTest/Hardware.hw

### AlarmMgr.vvm - PC_any/UnitTest/AlarmMgr.vvm
```iecst
(*Inputs to the unit test*)
VAR_CONFIG
	::AlarmMgr:MpAlarmXCoreMain.StatusID AT %Q.::AlarmXUnit:MpBlockStatus[0]; (*Insert your comment here...*)
	::AlarmMgr:MpAlarmXHistoryMain.StatusID AT %Q.::AlarmXUnit:MpBlockStatus[1]; (*Insert your comment here...*)
	::AlarmMgr:MpAlarmXHistoryUIMain.StatusID AT %Q.::AlarmXUnit:MpBlockStatus[2]; (*Insert your comment here...*)
	::AlarmMgr:MpAlarmXControlExample.StatusID AT %Q.::AlarmXUnit:MpBlockStatus[3]; (*Insert your comment here...*)
	::AlarmMgr:MpAlarmXListUIMain.StatusID AT %Q.::AlarmXUnit:MpBlockStatus[4]; (*Insert your comment here...*)
	::AlarmMgr:QueryActiveAlarms.StatusID AT %Q.::AlarmXUnit:MpBlockStatus[5]; (*Insert your comment here...*)
	::AlarmMgr:MpAlarmXCoreMain AT %Q.::AlarmXUnit:MpAlarmXCoreMain; (*Insert your comment here...*)
	::AlarmMgr:MpAlarmXListUIConnect AT %Q.::AlarmXUnit:MpAlarmXListUIConnect; (*Insert your comment here...*)
END_VAR
(*Outputs from the unit test*)
VAR_CONFIG
	::AlarmXUnit:AlarmExamples AT %Q.::AlarmMgr:AlarmExamples; (*Insert your comment here...*)
END_VAR
```

### AppAxis.vvm - PC_any/UnitTest/AppAxis.vvm
```iecst
(*Inputs to the unit test*)
VAR_CONFIG
	::AppAxis_1:MpAxisBasicAppAxis.StatusID AT %Q.::AppAxisUni:MpBlockStatus[0]; (*Insert your comment here...*)
	::AppAxis_1:MpAlarmXCoreAxis.StatusID AT %Q.::AppAxisUni:MpBlockStatus[1]; (*Insert your comment here...*)
	::AppAxis_1:MpRecipeRegParCfg.StatusID AT %Q.::AppAxisUni:MpBlockStatus[2]; (*Insert your comment here...*)
	::AppAxis_1:MpRecipeRegParPar.StatusID AT %Q.::AppAxisUni:MpBlockStatus[3]; (*Insert your comment here...*)
	::AppAxis_1:AxisControl.Status AT %Q.::AppAxisUni:AxisControl.Status; (*Insert your comment here...*)
	::AppAxis_1:MpAlarmXCoreAxis AT %Q.::AppAxisUni:MpAlarmXCoreAxis; (*Insert your comment here...*)
	::AppAxis_1:State AT %Q.::AppAxisUni:State; (*Insert your comment here...*)
END_VAR
(*Outputs from the unit test*)
VAR_CONFIG
	::AppAxisUni:AxisControl.Command AT %Q.::AppAxis_1:AxisControl.Command; (*Insert your comment here...*)
	::AppAxisUni:AxisControl.Parameters AT %Q.::AppAxis_1:AxisControl.Parameters; (*Insert your comment here...*)
END_VAR
```

### AuditMgr.vvm - PC_any/UnitTest/AuditMgr.vvm
```iecst
(*Inputs to the unit test*)
VAR_CONFIG
	::AuditMgr:MpAuditTrailSys.CommandDone AT %Q.::AuditTest:MpAuditTrailCmdDone; (*Insert your comment here...*)
	::AuditMgr:HmiAudit.Status.ArchiveAvailable AT %Q.::AuditTest:HmiAudit.Status.ArchiveAvailable; (*Insert your comment here...*)
	::AuditMgr:HmiAudit.Status.NumberOfArchives AT %Q.::AuditTest:HmiAudit.Status.NumberOfArchives; (*Insert your comment here...*)
	::AuditMgr:MpAuditTrailSys.Error AT %Q.::AuditTest:MpAuditTrailError; (*Insert your comment here...*)
END_VAR
(*Outputs from the unit test*)
VAR_CONFIG
	::AuditTest:HmiAudit.Commands.ExportArchives AT %Q.::AuditMgr:HmiAudit.Commands.ExportArchives; (*Insert your comment here...*)
	::AuditTest:SampleTemperature AT %Q.::AuditMgr:VariableMonitorExample; (*Insert your comment here...*)
	::AuditTest:HmiAudit.Parameters.ArchiveSettings.Enable AT %Q.::AuditMgr:HmiAudit.Parameters.ArchiveSettings.Enable; (*Insert your comment here...*)
	::AuditTest:HmiAudit.Parameters.ArchiveSettings.MaxSize AT %Q.::AuditMgr:HmiAudit.Parameters.ArchiveSettings.MaxSize; (*Insert your comment here...*)
	::AuditTest:HmiAudit.Parameters.ArchiveSettings.Mode AT %Q.::AuditMgr:HmiAudit.Parameters.ArchiveSettings.Mode; (*Insert your comment here...*)
	::AuditTest:HmiAudit.Parameters.ArchiveSettings.Hour AT %Q.::AuditMgr:HmiAudit.Parameters.ArchiveSettings.Hour; (*Insert your comment here...*)
	::AuditTest:HmiAudit.Parameters.ArchiveSettings.Minute AT %Q.::AuditMgr:HmiAudit.Parameters.ArchiveSettings.Minute; (*Insert your comment here...*)
	::AuditTest:HmiAudit.Parameters.ArchiveSettings.FileType AT %Q.::AuditMgr:HmiAudit.Parameters.ArchiveSettings.FileType; (*Insert your comment here...*)
END_VAR
```

### BackupMgr.vvm - PC_any/UnitTest/BackupMgr.vvm
```iecst
VAR_CONFIG
	::BackupMgr:MpBackupCoreSys.StatusID AT %Q.::BackupUnit:MpBlockStatus[0]; (*Insert your comment here...*)
	::BackupMgr:MpBackupCoreConfigSys.StatusID AT %Q.::BackupUnit:MpBlockStatus[1]; (*Insert your comment here...*)
	::BackupMgr:MpFileManagerUIBackup.StatusID AT %Q.::BackupUnit:MpBlockStatus[2]; (*Insert your comment here...*)
	::BackupMgr:HmiBackup.Status AT %Q.::BackupUnit:HmiBackup.Status; (*Insert your comment here...*)
	::BackupUnit:HmiBackup.Commands AT %Q.::BackupMgr:HmiBackup.Commands; (*Insert your comment here...*)
	::BackupUnit:HmiBackup.Parameters AT %Q.::BackupMgr:HmiBackup.Parameters; (*Insert your comment here...*)
END_VAR
```

### FileMgr.vvm - PC_any/UnitTest/FileMgr.vvm
```iecst
(*Inputs to the unit test*)
VAR_CONFIG
	::FileMgr:MpFileManagerUISys.StatusID AT %Q.::FileTest:MpBlockStatus[0]; (*Insert your comment here...*)
	::FileMgr:MpFileManagerUI_FIFO.StatusID AT %Q.::FileTest:MpBlockStatus[1]; (*Insert your comment here...*)
	Cyclic#8.::FileMgr:HmiFile.Status AT %Q.Cyclic#8.::FileTest:HmiFile_UT.Status; (*Insert your comment here...*)
	::FileMgr:MpFileManagerUIConnect.File.List.Items AT %Q.::FileTest:MpFileManagerUIConnect.File.List.Items; (*Insert your comment here...*)
	::FileMgr:MpFileManagerUIConnect.Status AT %Q.::FileTest:MpFileManagerUIConnect.Status; (*Insert your comment here...*)
	::FileMgr:MpFileManagerUIConnect.File.PathInfo AT %Q.::FileTest:MpFileManagerUIConnect.File.PathInfo; (*Insert your comment here...*)
END_VAR
(*Outputs from the unit test*)
VAR_CONFIG
	Cyclic#8.::FileTest:HmiFile_UT.Parameters AT %Q.Cyclic#8.::FileMgr:HmiFile.Parameters; (*Insert your comment here...*)
	::FileTest:MpFileManagerUIConnect.DeviceList.SelectedIndex AT %Q.::FileMgr:MpFileManagerUIConnect.DeviceList.SelectedIndex; (*Insert your comment here...*)
	::FileTest:MpFileManagerUIConnect.File.NewName AT %Q.::FileMgr:MpFileManagerUIConnect.File.NewName; (*Insert your comment here...*)
	::FileTest:MpFileManagerUIConnect.File.CreateFolder AT %Q.::FileMgr:MpFileManagerUIConnect.File.CreateFolder; (*Insert your comment here...*)
	::FileTest:MpFileManagerUIConnect.File.Refresh AT %Q.::FileMgr:MpFileManagerUIConnect.File.Refresh; (*Insert your comment here...*)
	::FileTest:HmiFile.Status.SelectedIndex AT %Q.::FileMgr:HmiFile.Status.SelectedIndex; (*Insert your comment here...*)
	::FileTest:MpFileManagerUIConnect.File.Copy AT %Q.::FileMgr:MpFileManagerUIConnect.File.Copy; (*Insert your comment here...*)
	::FileTest:MpFileManagerUIConnect.File.Paste AT %Q.::FileMgr:MpFileManagerUIConnect.File.Paste; (*Insert your comment here...*)
	::FileTest:MpFileManagerUIConnect.File.Rename AT %Q.::FileMgr:MpFileManagerUIConnect.File.Rename; (*Insert your comment here...*)
	::FileTest:MpFileManagerUIConnect.File.Cut AT %Q.::FileMgr:MpFileManagerUIConnect.File.Cut; (*Insert your comment here...*)
	::FileTest:HmiFile.Commands.EnterFolder AT %Q.::FileMgr:HmiFile.Commands.EnterFolder; (*Insert your comment here...*)
	::FileTest:HmiFile.Commands.FolderUp AT %Q.::FileMgr:HmiFile.Commands.FolderUp; (*Insert your comment here...*)
	::FileTest:MpFileManagerUIConnect.File.MultiSelect AT %Q.::FileMgr:MpFileManagerUIConnect.File.MultiSelect; (*Insert your comment here...*)
	::FileTest:MpFileManagerUIConnect.File.List.Items[0].IsSelected AT %Q.::FileMgr:MpFileManagerUIConnect.File.List.Items[0].IsSelected; (*Insert your comment here...*)
	::FileTest:MpFileManagerUIConnect.File.List.Items[1].IsSelected AT %Q.::FileMgr:MpFileManagerUIConnect.File.List.Items[1].IsSelected; (*Insert your comment here...*)
	::FileTest:MpFileManagerUIConnect.File.Filter AT %Q.::FileMgr:MpFileManagerUIConnect.File.Filter; (*Insert your comment here...*)
	::FileTest:MpFileManagerUIConnect.File.SortOrder AT %Q.::FileMgr:MpFileManagerUIConnect.File.SortOrder; (*Insert your comment here...*)
	::FileTest:MpFileManagerUIConnect.File.Delete AT %Q.::FileMgr:MpFileManagerUIConnect.File.Delete; (*Insert your comment here...*)
	::FileTest:MpFileManagerUIConnect.MessageBox.Confirm AT %Q.::FileMgr:MpFileManagerUIConnect.MessageBox.Confirm; (*Insert your comment here...*)
END_VAR
```

### RecipeMgr.vvm - PC_any/UnitTest/RecipeMgr.vvm
```iecst
(*Inputs to the unit test*)
VAR_CONFIG
	::RecipeMgr:MpFileManagerUIRecipe.StatusID AT %Q.::RecipeMgrU:MpBlockStatus[0]; (*Insert your comment here...*)
	::RecipeMgr:MpRecipeSys.StatusID AT %Q.::RecipeMgrU:MpBlockStatus[1]; (*Insert your comment here...*)
	::RecipeMgr:MpRecipeRegPar_PreviewCfg.StatusID AT %Q.::RecipeMgrU:MpBlockStatus[2]; (*Insert your comment here...*)
	::RecipeMgr:MpRecipeRegPar_PreviewPar.StatusID AT %Q.::RecipeMgrU:MpBlockStatus[3]; (*Insert your comment here...*)
	::RecipeMgr:MpRecipeUISys.StatusID AT %Q.::RecipeMgrU:MpBlockStatus[4]; (*Insert your comment here...*)
	::RecipeMgr:MachineSettings AT %Q.::RecipeMgrU:MachineSettings; (*Insert your comment here...*)
	::RecipeMgr:Parameters AT %Q.::RecipeMgrU:Parameters; (*Insert your comment here...*)
	::RecipeMgr:HmiRecipe.Status AT %Q.::RecipeMgrU:HmiRecipe.Status; (*Insert your comment here...*)
	::RecipeMgr:MpRecipeSys AT %Q.::RecipeMgrU:MpRecipeSys; (*Insert your comment here...*)
	::RecipeMgr:MpRecipeUIConnect.Recipe.List.Names AT %Q.::RecipeMgrU:MpRecipeUIConnect.Recipe.List.Names; (*Insert your comment here...*)
	::RecipeMgr:ParametersPreview AT %Q.::RecipeMgrU:ParametersPreview; (*Insert your comment here...*)
	::RecipeMgr:MpRecipeUIConnect.Recipe.List.MaxSelection AT %Q.::RecipeMgrU:MpRecipeUIConnect.Recipe.List.MaxSelection; (*Insert your comment here...*)
	::RecipeMgr:MpRecipeUIConnect.Status AT %Q.::RecipeMgrU:MpRecipeUIConnect.Status; (*Insert your comment here...*)
	::RecipeMgr:MpRecipeUIConnect.MessageBox.LayerStatus AT %Q.::RecipeMgrU:MpRecipeUIConnect.MessageBox.LayerStatus; (*Insert your comment here...*)
END_VAR
(*Outputs from the unit test*)
VAR_CONFIG
	::RecipeMgrU:HmiRecipe.Commands AT %Q.::RecipeMgr:HmiRecipe.Commands; (*Insert your comment here...*)
	::RecipeMgrU:HmiRecipe.Parameters AT %Q.::RecipeMgr:HmiRecipe.Parameters; (*Insert your comment here...*)
	::RecipeMgrU:MpRecipeUIConnect.Recipe.Filter AT %Q.::RecipeMgr:MpRecipeUIConnect.Recipe.Filter; (*Insert your comment here...*)
	::RecipeMgrU:MpRecipeUIConnect.Recipe.Refresh AT %Q.::RecipeMgr:MpRecipeUIConnect.Recipe.Refresh; (*Insert your comment here...*)
	::RecipeMgrU:MpRecipeUIConnect.Recipe.Load AT %Q.::RecipeMgr:MpRecipeUIConnect.Recipe.Load; (*Insert your comment here...*)
	::RecipeMgrU:ParametersEdit AT %Q.::RecipeMgr:ParametersEdit; (*Insert your comment here...*)
	::RecipeMgrU:MpRecipeUIConnect.Recipe.Delete AT %Q.::RecipeMgr:MpRecipeUIConnect.Recipe.Delete; (*Insert your comment here...*)
	::RecipeMgrU:MpRecipeUIConnect.MessageBox.Confirm AT %Q.::RecipeMgr:MpRecipeUIConnect.MessageBox.Confirm; (*Insert your comment here...*)
	::RecipeMgrU:MpRecipeUIConnect.Recipe.List.SelectedIndex AT %Q.::RecipeMgr:MpRecipeUIConnect.Recipe.List.SelectedIndex; (*Insert your comment here...*)
END_VAR
```

### ReportMgr.vvm - PC_any/UnitTest/ReportMgr.vvm
```iecst
VAR_CONFIG
	::ReportMgr:MpFileManagerUIReport.StatusID AT %Q.::ReportUnit:MpBlockStatus[0]; (*Insert your comment here...*)
	Cyclic#8.::ReportUnit:HmiReport_UT.Commands AT %Q.Cyclic#8.::ReportMgr:HmiReport.Commands; (*Insert your comment here...*)
	Cyclic#8.::ReportUnit:HmiReport_UT.Parameters.UseAdvancedFormat AT %Q.Cyclic#8.::ReportMgr:HmiReport.Parameters.UseAdvancedFormat; (*Insert your comment here...*)
	Cyclic#8.::ReportMgr:HmiReport.Status AT %Q.Cyclic#8.::ReportUnit:HmiReport_UT.Status; (*Insert your comment here...*)
	Cyclic#8.::ReportMgr:MpReportCoreSys.Active AT %Q.::ReportUnit:CoreInfoActive; (*Insert your comment here...*)
	Cyclic#8.::ReportMgr:MpReportCoreSys.CommandDone AT %Q.::ReportUnit:CoreCmdDone; (*Insert your comment here...*)
	Cyclic#8.::ReportMgr:MpReportCoreSys.Info AT %Q.::ReportUnit:CoreInfo_UT; (*Insert your comment here...*)
END_VAR
```

## Logical view

Binary libraries used (declarations not repeated): operator, runtime, astime, AsIecCon, FileIO, AsBrStr, sys_lib, standard, AsZip, AsIODiag, AsUSB, MpServer 5.18.0, MpAlarmX 5.18.0, MpBase 5.18.0, MpUserX 5.18.0, MpBackup 5.18.0, MpFile 5.18.0, MpCom 5.18.0, MpRecipe 5.18.0, CoTrace 5.18.0, AsARCfg, MpAudit 5.18.0, MpReport 5.18.0, McBase 5.18.1, McAcpPar 5.18.1, McAcpAx 5.18.1, McAxis 5.18.1, MpAxis 5.18.1, McPureVAx 5.18.1, ArTextSys, AsBrWStr, AsTCP, ArEventLog, MpPackML 5.18.0, UtMgr 2.01.0, UtWs 2.01.0, snprintf 1.10.4

### Package Logical/Libraries - Global libraries

### Library Logical/Libraries/IecCheck (IEC) - Remember to remove this after testing!
Depends on: sys_lib, AsBrStr

#### IecCheck.fun - Exported functions and function blocks
```iecst
FUNCTION CheckDivSint : SINT (* Check divisor for SINT division *)
	VAR_INPUT
		divisor : SINT;
	END_VAR
END_FUNCTION

FUNCTION CheckDivUsint : USINT (* Check divisor for USINT division *)
	VAR_INPUT
		divisor : USINT;
	END_VAR
END_FUNCTION

FUNCTION CheckDivInt : INT (* Check divisor for INT division *)
	VAR_INPUT
		divisor : INT;
	END_VAR
END_FUNCTION

FUNCTION CheckDivUint : UINT (* Check divisor for UINT division *)
	VAR_INPUT
		divisor : UINT;
	END_VAR
END_FUNCTION

FUNCTION CheckDivDint : DINT (* Check divisor for DINT division *)
	VAR_INPUT
		divisor : DINT;
	END_VAR
END_FUNCTION

FUNCTION CheckDivUdint : UDINT (* Check divisor for UDINT division *)
	VAR_INPUT
		divisor : UDINT;
	END_VAR
END_FUNCTION

FUNCTION CheckDivReal : REAL (* Check divisor for REAL division *)
	VAR_INPUT
		divisor : REAL;
	END_VAR
END_FUNCTION

FUNCTION CheckDivLReal : LREAL (* Check divisor for LREAL division, not available for SG3 and SGC *)
	VAR_INPUT
		divisor : LREAL;
	END_VAR
END_FUNCTION

FUNCTION CheckBounds : DINT (* Check range for array access *)
	VAR_INPUT
		index : DINT;
		lower : DINT;
		upper : DINT;
	END_VAR
END_FUNCTION

FUNCTION CheckRange : DINT (* Check range for enumeration *)
	VAR_INPUT
		value : DINT;
		lower : DINT;
		upper : DINT;
	END_VAR
END_FUNCTION

FUNCTION CheckSignedSubrange : DINT (* Check range for subrange of signed data types *)
	VAR_INPUT
		value : DINT;
		lower : DINT;
		upper : DINT;
	END_VAR
END_FUNCTION

FUNCTION CheckUnsignedSubrange : UDINT (* Check range for subrange of unsigned data types *)
	VAR_INPUT
		value : UDINT;
		lower : UDINT;
		upper : UDINT;
	END_VAR
END_FUNCTION

FUNCTION CheckReadAccess : UDINT (* Check address when reading dynamic variables *)
	VAR_INPUT
		address : UDINT;
	END_VAR
END_FUNCTION

FUNCTION CheckWriteAccess : UDINT (* Check address when writing dynamic variables *)
	VAR_INPUT
		address : UDINT;
	END_VAR
END_FUNCTION

FUNCTION MakeEntry : UDINT (* Makes an entry (log book entry) in the error log book *)
	VAR
		taskname : STRING[30];
		group : USINT;
		status_name : UINT;
		out_text : STRING[80];
	END_VAR
	VAR_INPUT
		number : UINT;
		index : DINT;
		text : STRING[50];
	END_VAR
END_FUNCTION
```

#### IecCheck.st - Implementation file
```iecst
(* Check divisor for SINT division *)
FUNCTION CheckDivSint
	IF divisor=0 THEN
		CheckDivSint := 1;
		MakeEntry(55555, divisor, 'CheckDivSint');
	ELSE
		CheckDivSint := divisor;
	END_IF
END_FUNCTION

(* Check divisor for USINT division *)
FUNCTION CheckDivUsint
	IF divisor = 0 THEN
		CheckDivUsint := 1;
		MakeEntry(55555, divisor, 'CheckDivUsint');
	ELSE
		CheckDivUsint := divisor;
	END_IF
END_FUNCTION

(* Check divisor for INT division *)
FUNCTION CheckDivInt
	IF divisor = 0 THEN
		CheckDivInt := 1;
		MakeEntry(55555, divisor, 'CheckDivInt');
	ELSE
		CheckDivInt := divisor;
	END_IF
END_FUNCTION

(* Check divisor for UINT division *)
FUNCTION CheckDivUint
	IF divisor = 0 THEN
		CheckDivUint := 1;
		MakeEntry(55555, divisor, 'CheckDivUint');
	ELSE
		CheckDivUint := divisor;
	END_IF
END_FUNCTION

(* Check divisor for DINT division *)
FUNCTION CheckDivDint
	IF divisor = 0 THEN
		CheckDivDint := 1;
		MakeEntry(55555, divisor, 'CheckDivDint');
	ELSE
		CheckDivDint := divisor;
	END_IF
END_FUNCTION

(* Check divisor for UDINT division *)
FUNCTION CheckDivUdint
	IF divisor = 0 THEN
		CheckDivUdint := 1;
		MakeEntry(55555, divisor, 'CheckDivUdint');
	ELSE
		CheckDivUdint := divisor;
	END_IF
END_FUNCTION

(* Check divisor for REAL division *)
FUNCTION CheckDivReal
	IF divisor = 0 THEN
		CheckDivReal := 1;
		MakeEntry(55555, 0, 'CheckDivReal');
	ELSE
		CheckDivReal := divisor;
	END_IF
END_FUNCTION

(* Check divisor for LREAL division *)
FUNCTION CheckDivLReal
	IF divisor = 0 THEN
		CheckDivLReal := 1;
		MakeEntry(55555, 0, 'CheckDivLReal');
	ELSE
		CheckDivLReal := divisor;
	END_IF
END_FUNCTION

(* Check range for array access *)
FUNCTION CheckBounds
	IF index < lower THEN
		CheckBounds := lower;
		MakeEntry(55555, index, 'CheckBounds');
	ELSIF index > upper THEN
		CheckBounds := upper;
		MakeEntry(55555, index, 'CheckBounds');
	ELSE
		CheckBounds := index;
	END_IF
END_FUNCTION

(* Check range for enumeration *)
FUNCTION CheckRange
	IF value < lower THEN
		CheckRange := lower;
		MakeEntry(55555, value, 'CheckRange');
	ELSIF value > upper THEN
		CheckRange := upper;
		MakeEntry(55555, value, 'CheckRange');
	ELSE
		CheckRange := value;
	END_IF
END_FUNCTION

(* Check range for subrange of signed data types *)
FUNCTION CheckSignedSubrange
	IF value < lower THEN
		CheckSignedSubrange := lower;
		MakeEntry(55555, value, 'CheckSignedSubrange');
	ELSIF value > upper THEN
		CheckSignedSubrange := upper;
		MakeEntry(55555, value, 'CheckSignedSubrange');
	ELSE
		CheckSignedSubrange := value;
	END_IF
END_FUNCTION

(* Check range for subrange of unsigned data types *)
FUNCTION CheckUnsignedSubrange
	IF value < lower THEN
		CheckUnsignedSubrange := lower;
		MakeEntry(55555, value, 'CheckUnsignedSubrange');
	ELSIF value > upper THEN
		CheckUnsignedSubrange := upper;
		MakeEntry(55555, value, 'CheckUnsignedSubrange');
	ELSE
		CheckUnsignedSubrange := value;
	END_IF
END_FUNCTION

(* Check address when reading dynamic variables *)
FUNCTION CheckReadAccess
	IF address = 0 THEN
		(* TODO: Insert an appropriate code, see AutomationStudio help for further information *)
		MakeEntry(55555, address, 'Read from NULL');
	END_IF

	CheckReadAccess := 0;
END_FUNCTION

(* Check address when writing dynamic variables *)
FUNCTION CheckWriteAccess
	IF address = 0 THEN
		(* TODO: Insert an appropriate code, see AutomationStudio help for further information *)
		MakeEntry(55555, address, 'Write to NULL');
	END_IF

	CheckWriteAccess := 0;
END_FUNCTION

(* Makes an entry (log book entry) in the error log book *)
FUNCTION MakeEntry
	status_name := ST_name(0, ADR(taskname), ADR(group));
	brsstrcpy(ADR(out_text), ADR(text));
	brsstrcat(ADR(out_text), ADR(' > in task > '));
	brsstrcat(ADR(out_text), ADR(taskname));
	MakeEntry := ADR(out_text);
	ERRxwarning(number, index, ADR(out_text));
	// force page fault to get back trace
	brsmemcpy(0, 0, 1);
END_FUNCTION
```

### Library Logical/Libraries/LoggingLib (ANSIC, version 2.30.1)
Depends on: AsTCP, astime, FileIO, ArEventLog, snprintf, Runtime

#### LoggingLib.typ - Exported data types
```iecst
(********************************************************************
 * COPYRIGHT -- Bernecker + Rainer
 ********************************************************************
 * Library: AsLogger
 * File: AsLogger.typ
 * Author: buchananw
 * Created: August 19, 2009
 ********************************************************************
 * Data types of library AsLogger
 ********************************************************************)

TYPE
	LogStatus :
		(
		LOG_OK,
		LOG_NOT_VALID,
		LOG_ILLEGAL_LEVEL,
		LOG_INVALID_ARGUMENTS,
		LOG_DUPLICATE,
		LOG_BUSY := 65535
		);
	LogLevel :
		(
		LOG_LEVEL_DEBUG,
		LOG_LEVEL_INFO,
		LOG_LEVEL_WARN,
		LOG_LEVEL_ERROR,
		LOG_LEVEL_FATAL
		);
	ClientStatus_typ :
		(
		CLIENT_NOT_USED,
		CLIENT_PENDING,
		CLIENT_SENDING,
		CLIENT_DONE,
		CLIENT_DROPPING
		);
	LoggerClient_typ : 	STRUCT
		ident : UDINT;
		ipAddress : STRING[15];
		port : UINT;
		status : ClientStatus_typ;
		wouldBlockCount : USINT;
		close : TcpClose;
		send : TcpSend;
	END_STRUCT;
	AS_LOGGER_ERRORS :
		(
		ASLOGGER_INTERNAL_ERROR := 30000,
		ASLOGGER_ILLEGAL_FILENAME := 33000,
		ASLOGGER_ILLEGAL_DEVICENAME
		);
	AsLoggerServerInternal_typ : 	STRUCT
		state : USINT;
		ident : UDINT;
		open : TcpOpen;
		close : TcpClose;
		server : TcpServer;
		clientsActive : USINT;
		clients : ARRAY[0..7]OF LoggerClient_typ;
		outputIndex : UINT;
		sendBuffer : STRING[5000];
		sendBufferUsed : UINT;
	END_STRUCT;
	AsLoggerFileInternal_typ : 	STRUCT
		state : AS_FILE_LOGGER_STATE;
		fileNumber : USINT;
		fileOffset : UDINT;
		tempFileName : STRING[80];
		oldFileName : STRING[80];
		newFileName : STRING[80];
		tempString : STRING[500];
		outputIndex : UINT;
		FileCreate_0 : FileCreate;
		FileOpen_0 : FileOpen;
		FileClose_0 : FileClose;
		FileWrite_0 : FileWrite;
		FileCopy_0 : FileCopy;
		FileDelete_0 : FileDelete;
		writeBuffer : STRING[10000];
		writeBufferUsed : UINT;
	END_STRUCT;
	AsLoggerLogBookInternal_typ : 	STRUCT
		outputIndex : UINT;
		ArEventLogWrite_0 : ArEventLogWrite;
		ArEventLogGetIdent_0 : ArEventLogGetIdent;
		outputIndexRegistered : BOOL;
	END_STRUCT;
	AS_FILE_LOGGER_STATE :
		(
		AS_FILE_LOGGER_STATE_W_ENABLE,
		AS_FILE_LOGGER_STATE_MOVE_FILES,
		AS_FILE_LOGGER_STATE_DELETE_OLD,
		AS_FILE_LOGGER_STATE_CREATE_FILE,
		AS_FILE_LOGGER_STATE_MARSHALL,
		AS_FILE_LOGGER_STATE_OPEN,
		AS_FILE_LOGGER_STATE_WRITE,
		AS_FILE_LOGGER_STATE_CLOSE,
		AS_FILE_LOGGER_STATE_ERROR := 255
		);
END_TYPE
```

#### LoggingLib.var - Exported constants
```iecst
(********************************************************************
 * COPYRIGHT -- Bernecker + Rainer
 ********************************************************************
 * Library: AsLogger
 * File: AsLogger.var
 * Author: buchananw
 * Created: August 19, 2009
 ********************************************************************
 * Constants of library AsLogger
 ********************************************************************)
VAR CONSTANT
	LOGGING_MAX_ARGUMENTS : USINT := 8;
END_VAR
```

#### LoggingLib.fun - Exported functions and function blocks
```iecst
(********************************************************************
 * COPYRIGHT -- Bernecker + Rainer
 ********************************************************************
 * Library: AsLogger
 * File: AsLogger.fun
 * Author: buchananw
 * Created: August 19, 2009
 ********************************************************************
 * Functions and function blocks of library AsLogger
 ********************************************************************)

FUNCTION logDebug : LogStatus
	VAR_INPUT
		name : STRING[80];
		message : STRING[256];
		pMsgData : UDINT;
	END_VAR
END_FUNCTION

FUNCTION logInfo : LogStatus
	VAR_INPUT
		name : STRING[80];
		message : STRING[256];
		pMsgData : UDINT;
	END_VAR
END_FUNCTION

FUNCTION logWarn : LogStatus
	VAR_INPUT
		name : STRING[80];
		message : STRING[256];
		pMsgData : UDINT;
	END_VAR
END_FUNCTION

FUNCTION logError : LogStatus
	VAR_INPUT
		name : STRING[80];
		message : STRING[256];
		pMsgData : UDINT;
	END_VAR
END_FUNCTION

FUNCTION logFatal : LogStatus
	VAR_INPUT
		name : STRING[80];
		message : STRING[256];
		pMsgData : UDINT;
	END_VAR
END_FUNCTION

FUNCTION_BLOCK AsLoggerServer
	VAR_INPUT
		port : UINT;
		disconnect : BOOL;
		level : LogLevel;
	END_VAR
	VAR_OUTPUT
		status : UINT;
	END_VAR
	VAR
		internal : AsLoggerServerInternal_typ;
	END_VAR
END_FUNCTION_BLOCK

FUNCTION_BLOCK AsLoggerFile
	VAR_INPUT
		enable : BOOL;
		device : STRING[80];
		fileName : STRING[80];
		maxFileSize : UDINT;
		maxFiles : USINT;
		delimiter : STRING[2];
		fileExtension : STRING[4];
		level : LogLevel;
	END_VAR
	VAR_OUTPUT
		status : UINT;
	END_VAR
	VAR
		internal : AsLoggerFileInternal_typ;
	END_VAR
END_FUNCTION_BLOCK

FUNCTION_BLOCK AsLoggerLogBook
	VAR_INPUT
		level : LogLevel;
	END_VAR
	VAR_OUTPUT
		status : UINT;
	END_VAR
	VAR
		internal : AsLoggerLogBookInternal_typ;
	END_VAR
END_FUNCTION_BLOCK

FUNCTION AsLoggerGetLastMessage : UDINT (*Function mainly used for testing purposes*)
END_FUNCTION
```

#### LoggingLib.c
```c
/********************************************************************
 * COPYRIGHT -- Bernecker + Rainer
 ********************************************************************
 * Library: AsLogger
 * File: AsLogger.c
 * Author: buchananw
 * Created: August 19, 2009
 *******************************************************************/

#include <bur/plctypes.h>
#include <LoggingLib.h>
#include "AsLoggerInternal.h"
#include <string.h>
#include <stdbool.h>

static LogStore_typ LogStore;

LogStatus logDebug(char* name, char* message, UDINT pMsgData)
{
    return logMessage(name, LOG_LEVEL_DEBUG, message, pMsgData);
}

LogStatus logInfo(char* name, char* message, UDINT pMsgData)
{
    return logMessage(name, LOG_LEVEL_INFO, message, pMsgData);
}

LogStatus logWarn(char* name, char* message, UDINT pMsgData)
{
    return logMessage(name, LOG_LEVEL_WARN, message, pMsgData);
}

LogStatus logError(char* name, char* message, UDINT pMsgData)
{
    return logMessage(name, LOG_LEVEL_ERROR, message, pMsgData);
}

LogStatus logFatal(char* name, char* message, UDINT pMsgData)
{
    return logMessage(name, LOG_LEVEL_FATAL, message, pMsgData);
}

UDINT AsLoggerGetLastMessage(void)
{
    UINT lastMessage = LogStore.inputIndex;

    return (UDINT)&LogStore.messages[decrementIndex(lastMessage)].message;
}

BOOL logLevelIsValid(LogLevel level)
{
    return ((level >= LOG_LEVEL_DEBUG) && (level <= LOG_LEVEL_FATAL));
}

BOOL isSameAsLastMessage(char* name, const char* message)
{
    unsigned int i = 0;
    for (i=0; i<sizeof(LogStore.lastMessages)/sizeof(LogStore.lastMessages[0]); i++)
    {
        if ((strcmp(LogStore.lastMessages[i].name, name) == 0) && (strcmp(LogStore.lastMessages[i].message, message) == 0))
            return true;
    }

    // message not found
    for (i=0; i<sizeof(LogStore.lastMessages)/sizeof(LogStore.lastMessages[0]); i++)
    {
        if (strcmp(LogStore.lastMessages[i].name, "") == 0)
        {
            strcpy(LogStore.lastMessages[i].name, name);
        }
        if (strcmp(LogStore.lastMessages[i].name, name) == 0)
        {
            strcpy(LogStore.lastMessages[i].message, message);
            break;
        }
    }

    return false;
}

LogStatus logMessage(char* name, LogLevel level, const char* message, UDINT pMsgData)
{
    UINT tempIndex;
    UtcDTGetTime_typ now;
    UtcDTStructureGetTime_typ UtcDTStructureGetTime_0;
    DTStructure nowMilliseconds;

    STRING formattedMessage[MAX_MESSAGE_LENGTH];
    char* currentChar;
    USINT currentArgIndex;
    UDINT** pData;
    char* arguments[LOGGING_MAX_ARGUMENTS];
    char argumentsTemp[LOGGING_MAX_ARGUMENTS][80];
    char tempMessage[256];

    if (logLevelIsValid(level) == false)
    {
        return LOG_ILLEGAL_LEVEL;
    }

    if (name == NULL)
    {
        return LOG_INVALID_ARGUMENTS;
    }
    if (message == NULL)
    {
        return LOG_INVALID_ARGUMENTS;
    }

    if (pMsgData == (UDINT)NULL)
    {
        strcpy(formattedMessage, message);
    }
    else
    {
        currentArgIndex = 0;
        pData = (void*)pMsgData;
        memset(&argumentsTemp, 0, sizeof(argumentsTemp));
        memset(&arguments, 0, sizeof(arguments));
        memset(&tempMessage, 0, sizeof(tempMessage));
        strcpy(tempMessage, message);
        currentChar = (char*)&tempMessage;

        while ((*currentChar != '\0') && (currentArgIndex < LOGGING_MAX_ARGUMENTS))
        {
            if (*currentChar == '%')
            {
                char nextChar;
                if (pData[currentArgIndex] == 0)
                    return LOG_INVALID_ARGUMENTS;

                switch (*(++currentChar))
                {
                    case 'b':
                        if (*(BOOL*)(pData[currentArgIndex]) == true)
                            strcpy(argumentsTemp[currentArgIndex], "TRUE");
                        else
                            strcpy(argumentsTemp[currentArgIndex], "FALSE");
                        arguments[currentArgIndex] = (char*)argumentsTemp[currentArgIndex];
                        // change %b to %s since we are creating the string.
                        *(currentChar) = 's';
                        break;
                    case 'l':
                        nextChar = *(currentChar + 1);
                        switch (nextChar)
                        {
                            case 'i':
                            case 'd':
                                strcpy(currentChar, (currentChar + 1));
                                *(currentChar + strlen(currentChar)) = 0;
                                snprintf2(argumentsTemp[currentArgIndex], (sizeof(argumentsTemp[0]) / sizeof(argumentsTemp[0][0])) - 1, "%li", *(DINT*)pData[currentArgIndex]);
                            break;
                            case 'u':
                                strcpy(currentChar, (currentChar + 1));
                                *(currentChar + strlen(currentChar)) = 0;
                                snprintf2(argumentsTemp[currentArgIndex],(sizeof(argumentsTemp[0]) / sizeof(argumentsTemp[0][0])) - 1, "%lu", *(UDINT*)pData[currentArgIndex]);
                            break;
                            case 'f':
                                strcpy(currentChar, (currentChar + 1));
                                *(currentChar + strlen(currentChar)) = 0;
                                snprintf2(argumentsTemp[currentArgIndex],(sizeof(argumentsTemp[0]) / sizeof(argumentsTemp[0][0])) - 1, "%lf", *(LREAL*)pData[currentArgIndex]);
                            break;
                        }
                        arguments[currentArgIndex] = (char*)argumentsTemp[currentArgIndex];
                        // change %b to %s since we are creating the string.
                        *(currentChar) = 's';
                        break;
                    case 's':
                        if ((currentChar + 1) != 0)
                        {
                            nextChar = *(currentChar + 1);
                            switch (nextChar)
                            {
                                case 'i':
                                case 'd':
                                    strcpy(currentChar, (currentChar + 1));
                                    *(currentChar + strlen(currentChar)) = 0;
                                    snprintf2(argumentsTemp[currentArgIndex],(sizeof(argumentsTemp[0]) / sizeof(argumentsTemp[0][0])) - 1, "%i", *(SINT*)pData[currentArgIndex]);
                                    break;
                                case 'u':
                                    strcpy(currentChar, (currentChar + 1));
                                    *(currentChar + strlen(currentChar)) = 0;
                                    snprintf2(argumentsTemp[currentArgIndex],(sizeof(argumentsTemp[0]) / sizeof(argumentsTemp[0][0])) - 1, "%i", *(USINT*)pData[currentArgIndex]);
                                    break;
                                default:
                                    snprintf2(argumentsTemp[currentArgIndex],(sizeof(argumentsTemp[0]) / sizeof(argumentsTemp[0][0])) - 1, "%s", (char*)pData[currentArgIndex]);
                            }
                        }
                        arguments[currentArgIndex] = (char*)argumentsTemp[currentArgIndex];
                        // change %b to %s since we are creating the string.
                        *(currentChar) = 's';
                        break;
                    case 'd':
                    case 'i':
                        snprintf2(argumentsTemp[currentArgIndex],(sizeof(argumentsTemp[0]) / sizeof(argumentsTemp[0][0])) - 1, "%i", *(INT*)pData[currentArgIndex]);
                        arguments[currentArgIndex] = (char*)argumentsTemp[currentArgIndex];
                        // change %d to %s since we are creating the string.
                        *(currentChar) = 's';
                        break;
                    case 'u':
                        snprintf2(argumentsTemp[currentArgIndex],(sizeof(argumentsTemp[0]) / sizeof(argumentsTemp[0][0])) - 1, "%u", *(UINT*)pData[currentArgIndex]);
                        arguments[currentArgIndex] = (char*)argumentsTemp[currentArgIndex];
                        // change %d to %s since we are creating the string.
                        *(currentChar) = 's';
                        break;
                    case 'f':
                        snprintf2(argumentsTemp[currentArgIndex],(sizeof(argumentsTemp[0]) / sizeof(argumentsTemp[0][0])) - 1, "%f", *(REAL*)pData[currentArgIndex]);
                        arguments[currentArgIndex] = (char*)argumentsTemp[currentArgIndex];
                        // change %f to %s since we are creating the string.
                        *(currentChar) = 's';
                        break;
                    case '%':
                        // this isn't an argument index so make sure the index isn't incremented
                        currentArgIndex--;
                        break;
                }
                currentArgIndex++;
            }
            else
            {
                currentChar++;
            }
        }

        memset(&formattedMessage, 0, sizeof(formattedMessage));
        snprintf2(formattedMessage,(sizeof(formattedMessage) / sizeof(formattedMessage[0])) - 1, tempMessage, arguments[0], arguments[1], arguments[2], arguments[3], arguments[4], arguments[5], arguments[6], arguments[7]);
    }

    if (isSameAsLastMessage(name, formattedMessage) == true)
        return LOG_DUPLICATE;

    /* no need for a lock because we increment the input index before doing anything else */
    tempIndex = LogStore.inputIndex;
    incrementIndex(LogStore.inputIndex);

    /* if the log buffer is full than forget the old messages */
    updateOutputIndexes(LogStore.outputIndexes, LogStore.inputIndex);

    strncpy(LogStore.messages[tempIndex].name, name, (sizeof(LogStore.messages[tempIndex].name) / sizeof(LogStore.messages[tempIndex].name[0])) - 1);
    strncpy(LogStore.messages[tempIndex].message, formattedMessage, (sizeof(LogStore.messages[tempIndex].message) / sizeof(LogStore.messages[tempIndex].message[0])) - 1);

    LogStore.messages[tempIndex].level = level;

    now.enable = true;
    UtcDTGetTime(&now);
    LogStore.messages[tempIndex].timeStamp = now.DT1;
    UtcDTStructureGetTime_0.enable = true ;
    UtcDTStructureGetTime_0.pDTStructure = (UDINT)&nowMilliseconds;
    UtcDTStructureGetTime(&UtcDTStructureGetTime_0);
    LogStore.messages[tempIndex].timeStampMilliseconds = nowMilliseconds.millisec;
    LogStore.messages[tempIndex].used = true;

    return LOG_OK;
}

LogStore_typ* getLogStore(void)
{
    return &LogStore;
}

BOOL addNewOutputIndex(UINT* newOutputIndex)
{
    USINT i = 0;
    while ((LogStore.outputIndexes[i] != NULL) && (i < (sizeof(LogStore.outputIndexes)/sizeof(LogStore.outputIndexes[0]))))
    {
        i++;
    }
    if (LogStore.outputIndexes[i] == NULL)
    {
        LogStore.outputIndexes[i] = newOutputIndex;
        return true;
    }
    return false;
}

void updateOutputIndexes(UINT** outputIndexes, UINT inputIndex)
{
    USINT i=0;
    if (outputIndexes == NULL)
        return;

    for (i=0;i < (sizeof(LogStore.outputIndexes)/sizeof(LogStore.outputIndexes[0]));i++)
    {
        if ((outputIndexes[i] != NULL) && (*outputIndexes[i] == inputIndex))
        {
            incrementIndex(*outputIndexes[i]);
        }
    }
}
```

#### AsLoggerInternal.h
```c
/********************************************************************
 * COPYRIGHT -- Bernecker + Rainer
 ********************************************************************
 * Library: AsLogger
 * File: AsLoggerStructures.h
 * Author: buchananw
 * Created: August 19, 2009
 *******************************************************************/
#ifndef __AS_LOGGER_INTERNALS_H__
#define __AS_LOGGER_INTERNALS_H__

#include <bur/plctypes.h>
#include <LoggingLib.h>

//#define __DEBUG_LOGGING_LIBRARY__

#define MAX_LOG_ITEMS 255
#define MAX_MESSAGE_LENGTH 512
#define MAX_NAME_LENGTH 80
#define MAX_INDEXES 8

#define LOG_SEND_BUF_SIZE (sizeof(sendBuffer)/sizeof(sendBuffer[0]))
#define MAX_WOULD_BLOCK 25

#define incrementIndex(x) x = (x+1)%MAX_LOG_ITEMS
#define decrementIndex(x) x = (x > 0) ? x - 1 : MAX_LOG_ITEMS - 1

typedef struct LogMessage_typ
{
    BOOL used;
    STRING name[MAX_NAME_LENGTH];
    LogLevel level;
    DATE_AND_TIME timeStamp;
    USINT timeStampMilliseconds;
    STRING message[MAX_MESSAGE_LENGTH];
}LogMessage_typ;

typedef struct LastMessage_typ
{
    STRING name[MAX_NAME_LENGTH];
    STRING message[MAX_MESSAGE_LENGTH];
}LastMessage_typ;

typedef struct LogStore_typ
{
    UINT inputIndex;
    UINT* outputIndexes[MAX_INDEXES];
    LogLevel level;
    LogMessage_typ messages[MAX_LOG_ITEMS];
    LastMessage_typ lastMessages[30];
}LogStore_typ;

BOOL addNewOutputIndex(UINT* newOutputIndex);
void updateOutputIndexes(UINT** outputIndexes, UINT inputIndex);
LogStatus logMessage(char* name, LogLevel level, const char* message, UDINT pMsgData);
LoggerClient_typ* getNextFreeClient(struct AsLoggerServer* inst);
BOOL acceptClient(LoggerClient_typ* newClient, UDINT clientIdent, UINT clientPort);
BOOL freeClient(LoggerClient_typ* client);
BOOL dropClient(LoggerClient_typ* client);
void handleAllActiveClients(LoggerClient_typ* clients, USINT numberOfClients, USINT* activeClients, char* sendBuffer, UINT* sendBufferUsed, LogMessage_typ* messages, LogLevel level, UINT* outputIndex);
BOOL handleClient(LoggerClient_typ* client, char* sendBuffer, UINT sendBufferUsed);
void sendToClient(LoggerClient_typ* client, char* buffer, UINT bufferLength);
BOOL writeHeader(char* buffer, UINT* bufferPos);
BOOL writeFooter(char* buffer, UINT* bufferPos);
BOOL marchallLogMessageAsXML(char* buffer, UINT* bufferPos, LogMessage_typ* message);
void marshallBuffer(char* buffer, UINT* bufferPos, LogMessage_typ* messages, LogLevel level, UINT* outputIndex);
void marchallLogMessageForFile(LogMessage_typ* message, char* delimiter, char* tempString, UDINT sizeOfTempString);
void addStringToBuffer(char* buffer, UINT* bufferPos, char* newMessage);
USINT convertToArLogLevel(LogMessage_typ* message);

LogStore_typ* getLogStore(void);

#endif
```

#### AsLoggerServer.c
```c
/********************************************************************
 * COPYRIGHT -- Bernecker + Rainer
 ********************************************************************
 * Library: AsLogger
 * File: AsLoggerServer.c
 * Author: buchananw
 * Created: August 20, 2009
 *******************************************************************/

#include <bur/plctypes.h>
#include <LoggingLib.h>
#include <string.h>
#include <stdbool.h>
#include "AsLoggerInternal.h"

#define XMLHEADER "<?xml version=\"1.0\" encoding=\"utf-8\"?> <logReport version=\"1.0\">"
#define XMLFOOTER "</logReport>\r\n"
#define MAX_LOGS_AT_ONCE 5

void AsLoggerServer(struct AsLoggerServer* inst)
{
    LoggerClient_typ* newClient;
    LogStore_typ* logStore;
    BOOL clientStillActive = false;
    USINT i;
    UDINT arguments[LOGGING_MAX_ARGUMENTS];

    inst->status = LOG_BUSY;

    if (inst == NULL)
    {
        logError("AsLoggerServer", "AsLoggerServer called with NULL instance", (UDINT)NULL);
        return;
    }
    switch (inst->internal.state)
    {
        case  0 :
            inst->internal.open.enable = true;
            inst->internal.open.pIfAddr = (UDINT)NULL;
            inst->internal.open.port = inst->port;
            TcpOpen(&inst->internal.open);
            inst->status = inst->internal.open.status;
            if (inst->internal.open.status == 0)
            {
                addNewOutputIndex(&inst->internal.outputIndex);
                inst->internal.ident = inst->internal.open.ident;
                inst->internal.open.enable = false;
                inst->internal.state = 10;
            }
            break;

        case 10: /* accept clients in this state */
            if (inst->disconnect == true)
            {
                inst->internal.state = 20;
                return;
            }

            if (inst->internal.clientsActive > 0)
            {
                logStore = getLogStore();
                if (logStore == NULL)
                {
                    inst->status = 1;
                    return;
                }
                handleAllActiveClients(&inst->internal.clients[0], sizeof(inst->internal.clients)/sizeof(inst->internal.clients[0]), &inst->internal.clientsActive, (char*)&inst->internal.sendBuffer, &inst->internal.sendBufferUsed, &logStore->messages[0], inst->level, &inst->internal.outputIndex);
            }

            newClient = getNextFreeClient(inst);

            if (newClient == NULL)
            {
                return;
            }

            inst->internal.server.enable = true;
            inst->internal.server.ident = inst->internal.ident;
            inst->internal.server.pIpAddr = (UDINT)newClient->ipAddress;

            TcpServer(&inst->internal.server);
            inst->status = inst->internal.server.status;
            if (inst->internal.server.status == 0)
            {
                for (i=0;i<(sizeof(inst->internal.clients)/sizeof(inst->internal.clients[0]));i++)
                {
                    if ((&inst->internal.clients[i] != newClient) && (strcmp(inst->internal.clients[i].ipAddress, newClient->ipAddress) == 0) && (inst->internal.clients[i].status != CLIENT_NOT_USED))
                    {
                        freeClient(newClient);
                        return;
                    }
                }
                //snprintf2(logString, (sizeof(logString) / sizeof(logString[0])) - 1, "accepting new client %s", newClient->ipAddress);
                arguments[0] = (UDINT)newClient->ipAddress;
                logDebug("AsLoggerServer",  "accepting new client %s", (UDINT)&arguments);
                /* accept client */
                if (acceptClient(newClient, inst->internal.server.identclnt, inst->internal.server.portclnt) == true)
                    inst->internal.clientsActive++;
            }
            break;

        case 20: /* disconnect all clients */
            inst->status = LOG_BUSY;
            clientStillActive = false;
            for (i=0;i<(sizeof(inst->internal.clients)/sizeof(inst->internal.clients[0]));i++)
            {
                if (inst->internal.clients[i].status != CLIENT_NOT_USED)
                {
                    clientStillActive |= dropClient(&inst->internal.clients[i]);
                }
            }
            if (clientStillActive == false)
            {
                inst->internal.state = 22;
            }
            break;

        case 22:
            inst->internal.close.enable = true;
            inst->internal.close.how = 0;
            inst->internal.close.ident = inst->internal.ident;
            TcpClose(&inst->internal.close);
            inst->status = inst->internal.close.status;
            if (inst->internal.close.status != 65535)
            {
                inst->status = 0;
                inst->internal.state = 0;
            }
            break;

        default :
            /* do nothing */
            break;
    }
}

LoggerClient_typ* getNextFreeClient(struct AsLoggerServer* inst)
{
    USINT i;
    for (i = 0; i < (sizeof(inst->internal.clients)/sizeof(inst->internal.clients[0])); i++) {
        if (inst->internal.clients[i].status == CLIENT_NOT_USED)
        {
            return &inst->internal.clients[i];
        }
    }
    return NULL;
}

BOOL acceptClient(LoggerClient_typ* newClient, UDINT clientIdent, UINT clientPort)
{
    if (newClient == NULL)
        return false;

    newClient->status = CLIENT_PENDING;
    newClient->ident = clientIdent;
    newClient->port = clientPort;
    memset(&newClient->send, 0, sizeof(newClient->send));
    memset(&newClient->close, 0, sizeof(newClient->close));
    return true;
}

void sendToClient(LoggerClient_typ* client, char* buffer, UINT bufferLength)
{
    UDINT arguments[LOGGING_MAX_ARGUMENTS];

    if ((client == NULL) || (client->status == CLIENT_NOT_USED))
        return;

    client->send.enable = true;
    client->send.ident = client->ident;
    client->send.datalen = bufferLength;
    client->send.pData = (UDINT)buffer;
    client->send.flags = 0;

    client->status = CLIENT_SENDING;

    TcpSend(&client->send);

    if (client->send.status == 0)
    {
        client->wouldBlockCount = 0;
        client->status = CLIENT_DONE;
    }
    else if ((client->send.status == tcpERR_WOULDBLOCK) && (client->wouldBlockCount < MAX_WOULD_BLOCK))
    {
        client->wouldBlockCount++;
    }
    else if (client->send.status == tcpERR_SENTLEN)
    {
        /* try to send data again */
    }
    else if (client->send.status != 65535)
    {
        client->wouldBlockCount = 0;
        /* an error occured so drop the client */
        //snprintf2(errorString, (sizeof(errorString) / sizeof(errorString[0])) - 1, "error received while sending %d", client->send.status);
        arguments[0] = (UDINT)&client->send.status;
        logDebug("AsLoggerServer", "error received while sending %d", (UDINT)&arguments);
        client->status = CLIENT_DROPPING;
    }
}

BOOL dropClient(LoggerClient_typ* client)
{
    UDINT arguments[LOGGING_MAX_ARGUMENTS];
    if (client == NULL)
        return false;

    client->close.enable = true;
    client->close.ident = client->ident;
    client->close.how = 0;
    client->status = CLIENT_DROPPING;

    TcpClose(&client->close);
    if (client->close.status == 0)
    {
        //snprintf2(logString, (sizeof(logString) / sizeof(logString[0])) - 1, "dropped client %s", client->ipAddress);
        arguments[0] = (UDINT)&client->ipAddress;
        logDebug("AsLoggerServer", "dropped client %s", (UDINT)&arguments);
        return freeClient(client);
    }
    return false;
}

BOOL freeClient(LoggerClient_typ* client)
{
    if (client == NULL)
        return false;

    memset(client, 0, sizeof(*client));
    client->status = CLIENT_NOT_USED;
    return true;
}

BOOL handleClient(LoggerClient_typ* client, char* sendBuffer, UINT sendBufferUsed)
{
    if (client == NULL)
        return false;

    switch (client->status)
    {
        case CLIENT_NOT_USED:
        break;

        case CLIENT_PENDING:
        case CLIENT_SENDING:
            sendToClient(client, sendBuffer, sendBufferUsed);
        break;

        case CLIENT_DROPPING:
            return dropClient(client);
        break;

        case CLIENT_DONE:
            /* wait until all clients are finished sending before transitting out of the done state */
            /* handled by handleAllActiveClients */
        break;
    }
    return false;
}

void handleAllActiveClients(LoggerClient_typ* clients, USINT numberOfClients, USINT* activeClients, char* sendBuffer, UINT* sendBufferUsed, LogMessage_typ* messages, LogLevel level, UINT* outputIndex)
{
    USINT i;
    BOOL allClientsFinishedSending = true;

    for (i=0;i<numberOfClients;i++)
    {
        if ((clients[i].status == CLIENT_PENDING) || (clients[i].status == CLIENT_SENDING))
            allClientsFinishedSending = false;
    }

    if (allClientsFinishedSending == true)
    {
        for (i=0;i<numberOfClients;i++)
        {
            if (clients[i].status == CLIENT_DONE)
            {
                clients[i].status = CLIENT_PENDING;
            }
        }
        marshallBuffer(sendBuffer, sendBufferUsed, messages, level, outputIndex);
    }

    for (i=0;i<numberOfClients;i++)
    {
        if (clients[i].status != CLIENT_NOT_USED)
        {
            if (handleClient(&clients[i], sendBuffer, *sendBufferUsed) == true)
            {
                *activeClients = *activeClients - 1;
            }
        }
    }
}

void marshallBuffer(char* buffer, UINT* bufferPos, LogMessage_typ* messages, LogLevel level, UINT* outputIndex)
{
    USINT i;
    USINT numberOfLogs = 0;
    LogStore_typ* logStore = getLogStore();

    if ((buffer == NULL) || (bufferPos == NULL) || (messages == NULL) || (logStore == NULL))
        return;

    *bufferPos = 0;
    writeHeader(buffer, bufferPos);

    for (i=*outputIndex; (i != logStore->inputIndex) && (numberOfLogs < MAX_LOGS_AT_ONCE); incrementIndex(i))
    {
        if (messages[i].level >= level)
        {
            marchallLogMessageAsXML(buffer, bufferPos, &messages[i]);
        }
        incrementIndex(*outputIndex);
        numberOfLogs++;
    }
    writeFooter(buffer, bufferPos);

}

BOOL writeHeader(char* buffer, UINT* bufferPos)
{
    if ((buffer == NULL) || (bufferPos == NULL))
        return 0;

    strcpy((char*)buffer, XMLHEADER);
    *bufferPos = *bufferPos + strlen(XMLHEADER);
    return true;
}

BOOL writeFooter(char* buffer, UINT* bufferPos)
{
    strcpy((char*)(buffer + *bufferPos), XMLFOOTER);
    *bufferPos = *bufferPos + strlen(XMLFOOTER);
    return true;
}

BOOL marchallLogMessageAsXML(char* buffer, UINT* bufferPos, LogMessage_typ* message)
{
    STRING level[6];
    STRING tempString[900];

    if ((buffer == NULL) || (bufferPos == NULL) || (message == NULL))
        return false;

    switch(message->level)
    {
        case LOG_LEVEL_DEBUG:
            strcpy(level, "DEBUG");
        break;
        case LOG_LEVEL_INFO:
            strcpy(level, "INFO");
        break;
        case LOG_LEVEL_WARN:
            strcpy(level, "WARN");
        break;
        case LOG_LEVEL_ERROR:
            strcpy(level, "ERROR");
        break;
        case LOG_LEVEL_FATAL:
            strcpy(level, "FATAL");
        break;
    }

    snprintf2(tempString, (sizeof(tempString) / sizeof(tempString[0])) - 1, \
            "<logItem><log><![CDATA[AsLoggerServer]]></log><level>%s</level><date>%u</date><millis>%u</millis><taskName>%s</taskName><message><![CDATA[%s]]></message></logItem>", \
            level, message->timeStamp, message->timeStampMilliseconds, message->name, message->message);
    memcpy(buffer + *bufferPos, tempString, strlen(tempString));
    *bufferPos = *bufferPos + strlen(tempString);
    return true;
}
```
